Yaskawa INFORM job: pointsclTRJ2.JBI

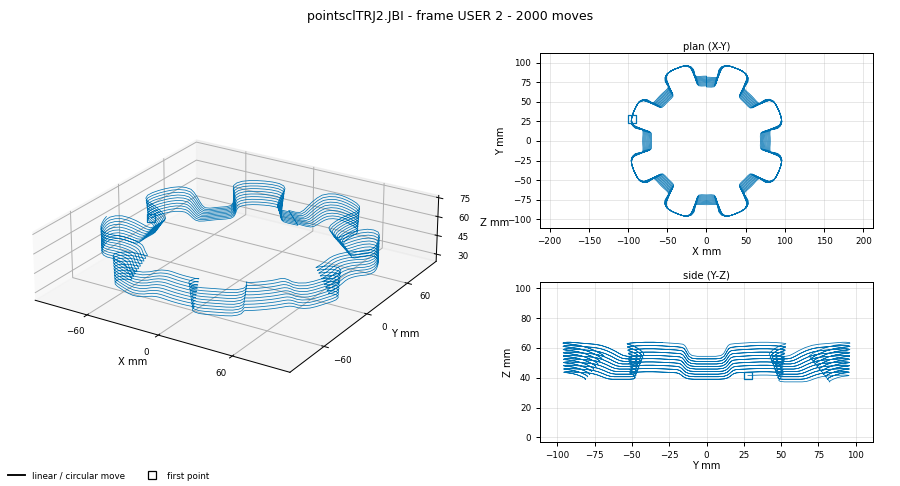
[picture p0: tool path of pointsclTRJ2.JBI in frame USER 2, 2000 of 2000 moves have a stored position in this frame; points joined in program order, loops and branches not executed]
/JOB
//NAME pointsclTRJ2
//POS
///NPOS 2000,0,0,0,0,0
///USER 2
///TOOL 1
///POSTYPE USER
///RECTAN
///RCONF 1,0,0,0,0,0,0,0,0,0,0,0,0,0,0,0,0,0,0,0,0,0,0,0
C00000=-95.500,27.752,41.515,166.5415,13.7835,0.0000
C00001=-94.679,31.992,41.678,168.5942,9.8161,0.0000
C00002=-93.214,36.189,41.785,170.1405,7.6437,0.0000
C00003=-91.502,40.323,41.785,-167.6355,-1.4870,0.0000
C00004=-89.570,44.326,41.678,-165.0261,-0.9876,0.0000
C00005=-87.153,47.905,41.515,-160.8334,0.4949,0.0000
C00006=-83.964,50.341,41.355,-155.1452,4.3197,0.0000
C00007=-80.606,51.270,41.159,-151.1279,10.7556,0.0000
C00008=-77.545,50.645,40.789,-149.8656,15.0064,0.0000
C00009=-74.511,49.565,40.048,-149.4700,17.9765,0.0000
C00010=-71.724,48.673,39.090,-149.4755,20.2620,0.0000
C00011=-69.261,48.447,38.165,-149.7708,22.3484,0.0000
C00012=-66.868,49.465,37.495,-150.5123,24.7951,0.0000
C00013=-64.059,52.288,37.229,-151.9366,27.5294,0.0000
C00014=-61.349,55.398,37.217,-151.9559,27.7386,0.0000
C00015=-58.451,58.451,37.225,-150.5381,26.1896,0.0000
C00016=-55.398,61.349,37.217,-149.2124,24.5903,0.0000
C00017=-52.288,64.059,37.229,-149.4318,24.6574,0.0000
C00018=-49.465,66.868,37.495,-152.0451,26.5426,0.0000
C00019=-48.447,69.261,38.165,-154.5539,27.7518,0.0000
C00020=-48.673,71.724,39.090,-156.8022,28.4553,0.0000
C00021=-49.565,74.511,40.048,-159.3588,28.8937,0.0000
C00022=-50.645,77.545,40.789,-162.7782,29.0063,0.0000
C00023=-51.270,80.606,41.159,-167.7607,28.3185,0.0000
C00024=-50.341,83.964,41.355,-175.2412,24.7794,0.0000
C00025=-47.905,87.153,41.515,-179.4760,19.1659,0.0000
C00026=-44.326,89.570,41.678,178.9776,14.9716,0.0000
C00027=-40.323,91.502,41.785,178.4777,12.3603,0.0000
C00028=-36.189,93.214,41.785,-172.2431,-9.7711,0.0000
C00029=-31.992,94.679,41.678,-169.9901,-11.2367,0.0000
C00030=-27.752,95.500,41.515,-165.8427,-13.0639,0.0000
C00031=-23.775,94.968,41.355,-158.8727,-14.0699,0.0000
C00032=-20.743,93.250,41.159,-151.4855,-11.7399,0.0000
C00033=-19.021,90.644,40.789,-147.8038,-9.1945,0.0000
C00034=-17.640,87.735,40.048,-145.6522,-7.0900,0.0000
C00035=-16.299,85.134,39.090,-144.2478,-5.2806,0.0000
C00036=-14.718,83.232,38.165,-143.1858,-3.4622,0.0000
C00037=-12.305,82.260,37.495,-142.2198,-1.1140,0.0000
C00038=-8.324,82.270,37.229,-141.5279,1.8234,0.0000
C00039=-4.208,82.553,37.217,-141.4104,1.9981,0.0000
C00040=0.000,82.662,37.225,-141.3795,0.0003,0.0000
C00041=0.000,81.307,38.958,-141.1409,0.0002,0.0000
C00042=4.084,81.202,38.949,-141.1716,-1.9954,0.0000
C00043=8.115,80.931,38.962,-141.2889,-1.7381,0.0000
C00044=12.050,80.963,39.253,-141.9942,1.3169,0.0000
C00045=14.402,82.041,39.987,-142.9610,3.6876,0.0000
C00046=15.932,84.113,41.004,-144.0223,5.5238,0.0000
C00047=17.234,86.943,42.060,-145.4570,7.3915,0.0000
C00048=18.580,90.119,42.880,-147.7223,9.6046,0.0000
C00049=20.259,92.987,43.289,-151.7341,12.2844,0.0000
C00050=23.317,94.913,43.506,-160.1091,14.4794,0.0000
C00051=27.389,95.566,43.684,-167.4562,12.7995,0.0000
C00052=31.762,94.755,43.864,-171.4202,10.6129,0.0000
C00053=36.110,93.244,43.984,-173.4230,9.0647,0.0000
C00054=40.400,91.468,43.984,178.1652,-11.0336,0.0000
C00055=44.543,89.461,43.864,178.4356,-13.5277,0.0000
C00056=48.209,86.942,43.684,179.5849,-17.8430,0.0000
C00057=50.626,83.601,43.506,-176.4717,-24.1883,0.0000
C00058=51.426,80.077,43.289,-168.3941,-28.5314,0.0000
C00059=50.586,76.861,42.880,-163.0330,-29.3601,0.0000
C00060=49.291,73.664,42.060,-159.4239,-29.2475,0.0000
C00061=48.211,70.742,41.004,-156.7894,-28.7861,0.0000
C00062=47.828,68.195,39.987,-154.5220,-28.0686,0.0000
C00063=48.729,65.770,39.253,-151.9898,-26.8420,0.0000
C00064=51.488,62.965,38.962,-149.2803,-24.8706,0.0000
C00065=54.531,60.307,38.949,-149.0055,-24.7373,0.0000
C00066=57.493,57.493,38.958,-150.3287,-26.3368,0.0000
C00067=60.306,54.531,38.949,-151.7425,-27.8849,0.0000
C00068=62.965,51.488,38.962,-151.6647,-27.6101,0.0000
C00069=65.770,48.729,39.253,-150.1785,-24.7729,0.0000
C00070=68.195,47.828,39.987,-149.4302,-22.3072,0.0000
C00071=70.742,48.211,41.004,-149.1281,-20.2070,0.0000
C00072=73.664,49.291,42.060,-149.1154,-17.8577,0.0000
C00073=76.861,50.586,42.880,-149.5380,-14.7348,0.0000
C00074=80.077,51.426,43.289,-150.9692,-10.1806,0.0000
C00075=83.601,50.626,43.506,-155.7711,-3.2182,0.0000
C00076=86.942,48.209,43.684,-162.1566,0.3951,0.0000
C00077=89.461,44.543,43.864,-166.4674,1.5210,0.0000
C00078=91.468,40.400,43.984,-168.9609,1.8009,0.0000
C00079=93.244,36.110,43.984,170.8762,-6.4945,0.0000
C00080=94.755,31.762,43.864,169.2698,-8.4320,0.0000
C00081=95.566,27.389,43.684,166.8982,-12.2272,0.0000
C00082=94.913,23.317,43.506,164.6442,-19.2338,0.0000
C00083=92.987,20.259,43.289,166.1133,-27.5629,0.0000
C00084=90.119,18.580,42.880,168.6818,-31.7718,0.0000
C00085=86.943,17.234,42.060,171.0499,-34.2159,0.0000
C00086=84.113,15.932,41.004,173.1852,-35.7848,0.0000
C00087=82.041,14.402,39.987,175.3839,-36.9495,0.0000
C00088=80.963,12.050,39.253,178.3288,-37.9940,0.0000
C00089=80.931,8.115,38.962,-177.7730,-38.6900,0.0000
C00090=81.202,4.084,38.949,-177.4393,-38.8004,0.0000
C00091=81.307,0.000,38.958,179.9997,-38.8591,0.0000
C00092=81.202,-4.084,38.949,177.4397,-38.8005,0.0000
C00093=80.931,-8.116,38.962,177.7742,-38.6899,0.0000
C00094=80.963,-12.050,39.253,-178.3283,-37.9939,0.0000
C00095=82.041,-14.402,39.987,-175.3840,-36.9495,0.0000
C00096=84.113,-15.932,41.004,-173.1855,-35.7848,0.0000
C00097=86.943,-17.234,42.060,-171.0504,-34.2160,0.0000
C00098=90.119,-18.580,42.880,-168.6823,-31.7720,0.0000
C00099=92.987,-20.259,43.289,-166.1135,-27.5630,0.0000
C00100=94.913,-23.317,43.506,-164.6442,-19.2338,0.0000
C00101=95.566,-27.389,43.684,-166.8982,-12.2272,0.0000
C00102=94.755,-31.762,43.864,-169.2698,-8.4320,0.0000
C00103=93.244,-36.110,43.984,-170.8762,-6.4945,0.0000
C00104=91.468,-40.400,43.984,168.9609,1.8009,0.0000
C00105=89.461,-44.543,43.864,166.4674,1.5210,0.0000
C00106=86.942,-48.209,43.684,162.1566,0.3951,0.0000
C00107=83.601,-50.626,43.506,155.7711,-3.2182,0.0000
C00108=80.077,-51.426,43.289,150.9692,-10.1803,0.0000
C00109=76.861,-50.586,42.880,149.5378,-14.7344,0.0000
C00110=73.664,-49.291,42.060,149.1152,-17.8573,0.0000
C00111=70.742,-48.211,41.004,149.1280,-20.2068,0.0000
C00112=68.195,-47.828,39.987,149.4301,-22.3071,0.0000
C00113=65.770,-48.729,39.253,150.1787,-24.7733,0.0000
C00114=62.965,-51.488,38.962,151.6652,-27.6109,0.0000
C00115=60.307,-54.531,38.949,151.7428,-27.8851,0.0000
C00116=57.493,-57.493,38.958,150.3283,-26.3364,0.0000
C00117=54.531,-60.306,38.949,149.0057,-24.7376,0.0000
C00118=51.488,-62.965,38.962,149.2810,-24.8713,0.0000
C00119=48.729,-65.770,39.253,151.9902,-26.8422,0.0000
C00120=47.828,-68.195,39.987,154.5219,-28.0685,0.0000
C00121=48.211,-70.742,41.004,156.7892,-28.7859,0.0000
C00122=49.291,-73.664,42.060,159.4235,-29.2473,0.0000
C00123=50.586,-76.861,42.880,163.0325,-29.3600,0.0000
C00124=51.426,-80.077,43.289,168.3938,-28.5314,0.0000
C00125=50.626,-83.601,43.506,176.4717,-24.1883,0.0000
C00126=48.209,-86.942,43.684,-179.5849,-17.8430,0.0000
C00127=44.543,-89.461,43.864,-178.4356,-13.5277,0.0000
C00128=40.400,-91.468,43.984,-178.1652,-11.0336,0.0000
C00129=36.110,-93.244,43.984,173.4230,9.0647,0.0000
C00130=31.762,-94.755,43.864,171.4202,10.6129,0.0000
C00131=27.389,-95.566,43.684,167.4562,12.7995,0.0000
C00132=23.317,-94.913,43.506,160.1091,14.4794,0.0000
C00133=20.259,-92.987,43.289,151.7341,12.2844,0.0000
C00134=18.580,-90.119,42.880,147.7223,9.6046,0.0000
C00135=17.234,-86.943,42.060,145.4570,7.3915,0.0000
C00136=15.932,-84.113,41.004,144.0223,5.5238,0.0000
C00137=14.402,-82.041,39.987,142.9610,3.6876,0.0000
C00138=12.050,-80.963,39.253,141.9942,1.3169,0.0000
C00139=8.115,-80.931,38.962,141.2889,-1.7381,0.0000
C00140=4.084,-81.202,38.949,141.1716,-1.9954,0.0000
C00141=0.000,-81.307,38.958,141.1409,0.0002,0.0000
C00142=0.000,-81.307,38.958,141.1409,0.0002,0.0000
C00143=-4.084,-81.202,38.949,141.1716,1.9951,0.0000
C00144=-8.116,-80.931,38.962,141.2890,1.7371,0.0000
C00145=-12.050,-80.963,39.253,141.9943,-1.3173,0.0000
C00146=-14.402,-82.041,39.987,142.9611,-3.6875,0.0000
C00147=-15.932,-84.113,41.004,144.0223,-5.5235,0.0000
C00148=-17.234,-86.943,42.060,145.4569,-7.3911,0.0000
C00149=-18.580,-90.119,42.880,147.7222,-9.6042,0.0000
C00150=-20.259,-92.987,43.289,151.7339,-12.2842,0.0000
C00151=-23.317,-94.913,43.506,160.1091,-14.4794,0.0000
C00152=-27.389,-95.566,43.684,167.4562,-12.7995,0.0000
C00153=-31.762,-94.755,43.864,171.4202,-10.6129,0.0000
C00154=-36.110,-93.244,43.984,173.4230,-9.0647,0.0000
C00155=-40.400,-91.468,43.984,-178.1652,11.0336,0.0000
C00156=-44.543,-89.461,43.864,-178.4356,13.5277,0.0000
C00157=-48.209,-86.942,43.684,-179.5849,17.8430,0.0000
C00158=-50.626,-83.601,43.506,176.4717,24.1883,0.0000
C00159=-51.426,-80.077,43.289,168.3941,28.5314,0.0000
C00160=-50.586,-76.861,42.880,163.0330,29.3601,0.0000
C00161=-49.291,-73.664,42.060,159.4239,29.2475,0.0000
C00162=-48.211,-70.742,41.004,156.7894,28.7861,0.0000
C00163=-47.828,-68.195,39.987,154.5220,28.0686,0.0000
C00164=-48.729,-65.770,39.253,151.9898,26.8420,0.0000
C00165=-51.488,-62.965,38.962,149.2803,24.8706,0.0000
C00166=-54.531,-60.307,38.949,149.0055,24.7373,0.0000
C00167=-57.493,-57.493,38.958,150.3287,26.3368,0.0000
C00168=-60.306,-54.531,38.949,151.7425,27.8849,0.0000
C00169=-62.965,-51.488,38.962,151.6647,27.6101,0.0000
C00170=-65.770,-48.729,39.253,150.1785,24.7729,0.0000
C00171=-68.195,-47.828,39.987,149.4302,22.3072,0.0000
C00172=-70.742,-48.211,41.004,149.1281,20.2070,0.0000
C00173=-73.664,-49.291,42.060,149.1154,17.8577,0.0000
C00174=-76.861,-50.586,42.880,149.5380,14.7348,0.0000
C00175=-80.077,-51.426,43.289,150.9692,10.1806,0.0000
C00176=-83.601,-50.626,43.506,155.7711,3.2182,0.0000
C00177=-86.942,-48.209,43.684,162.1566,-0.3951,0.0000
C00178=-89.461,-44.543,43.864,166.4674,-1.5210,0.0000
C00179=-91.468,-40.400,43.984,168.9609,-1.8009,0.0000
C00180=-93.244,-36.110,43.984,-170.8762,6.4945,0.0000
C00181=-94.755,-31.762,43.864,-169.2698,8.4320,0.0000
C00182=-95.566,-27.389,43.684,-166.8982,12.2272,0.0000
C00183=-94.913,-23.317,43.506,-164.6442,19.2338,0.0000
C00184=-92.987,-20.259,43.289,-166.1133,27.5629,0.0000
C00185=-90.119,-18.580,42.880,-168.6818,31.7718,0.0000
C00186=-86.943,-17.234,42.060,-171.0499,34.2159,0.0000
C00187=-84.113,-15.932,41.004,-173.1852,35.7848,0.0000
C00188=-82.041,-14.402,39.987,-175.3839,36.9495,0.0000
C00189=-80.963,-12.050,39.253,-178.3288,37.9940,0.0000
C00190=-80.931,-8.115,38.962,177.7730,38.6900,0.0000
C00191=-81.202,-4.084,38.949,177.4393,38.8004,0.0000
C00192=-81.307,0.000,38.958,-179.9997,38.8591,0.0000
C00193=-81.202,4.084,38.949,-177.4397,38.8005,0.0000
C00194=-80.931,8.116,38.962,-177.7742,38.6899,0.0000
C00195=-80.963,12.050,39.253,178.3283,37.9939,0.0000
C00196=-82.041,14.402,39.987,175.3840,36.9495,0.0000
C00197=-84.113,15.932,41.004,173.1855,35.7848,0.0000
C00198=-86.943,17.234,42.060,171.0504,34.2160,0.0000
C00199=-90.119,18.580,42.880,168.6823,31.7720,0.0000
C00200=-92.987,20.259,43.289,166.1135,27.5630,0.0000
C00201=-94.913,23.317,43.506,164.6442,19.2338,0.0000
C00202=-95.566,27.389,43.684,166.8982,12.2272,0.0000
C00203=-94.755,31.762,43.864,169.2698,8.4320,0.0000
C00204=-93.244,36.110,43.984,170.8762,6.4945,0.0000
C00205=-91.468,40.400,43.984,-168.9609,-1.8009,0.0000
C00206=-89.461,44.543,43.864,-166.4674,-1.5210,0.0000
C00207=-86.942,48.209,43.684,-162.1566,-0.3951,0.0000
C00208=-83.601,50.626,43.506,-155.7711,3.2182,0.0000
C00209=-80.077,51.426,43.289,-150.9692,10.1803,0.0000
C00210=-76.861,50.586,42.880,-149.5378,14.7344,0.0000
C00211=-73.664,49.291,42.060,-149.1152,17.8573,0.0000
C00212=-70.742,48.211,41.004,-149.1280,20.2068,0.0000
C00213=-68.195,47.828,39.987,-149.4301,22.3071,0.0000
C00214=-65.770,48.729,39.253,-150.1787,24.7733,0.0000
C00215=-62.965,51.488,38.962,-151.6652,27.6109,0.0000
C00216=-60.307,54.531,38.949,-151.7428,27.8851,0.0000
C00217=-57.493,57.493,38.958,-150.3283,26.3364,0.0000
C00218=-54.531,60.306,38.949,-149.0057,24.7376,0.0000
C00219=-51.488,62.965,38.962,-149.2810,24.8713,0.0000
C00220=-48.729,65.770,39.253,-151.9902,26.8422,0.0000
C00221=-47.828,68.195,39.987,-154.5219,28.0685,0.0000
C00222=-48.211,70.742,41.004,-156.7892,28.7859,0.0000
C00223=-49.291,73.664,42.060,-159.4235,29.2473,0.0000
C00224=-50.586,76.861,42.880,-163.0325,29.3600,0.0000
C00225=-51.426,80.077,43.289,-168.3938,28.5314,0.0000
C00226=-50.626,83.601,43.506,-176.4717,24.1883,0.0000
C00227=-48.209,86.942,43.684,179.5849,17.8430,0.0000
C00228=-44.543,89.461,43.864,178.4356,13.5277,0.0000
C00229=-40.400,91.468,43.984,178.1652,11.0336,0.0000
C00230=-36.110,93.244,43.984,-173.4230,-9.0647,0.0000
C00231=-31.762,94.755,43.864,-171.4202,-10.6129,0.0000
C00232=-27.389,95.566,43.684,-167.4562,-12.7995,0.0000
C00233=-23.317,94.913,43.506,-160.1091,-14.4794,0.0000
C00234=-20.259,92.987,43.289,-151.7339,-12.2842,0.0000
C00235=-18.580,90.119,42.880,-147.7222,-9.6042,0.0000
C00236=-17.234,86.943,42.060,-145.4569,-7.3911,0.0000
C00237=-15.932,84.113,41.004,-144.0223,-5.5235,0.0000
C00238=-14.402,82.041,39.987,-142.9611,-3.6875,0.0000
C00239=-12.050,80.963,39.253,-141.9943,-1.3173,0.0000
C00240=-8.116,80.931,38.962,-141.2890,1.7371,0.0000
C00241=-4.084,81.202,38.949,-141.1716,1.9951,0.0000
C00242=0.000,81.307,38.958,-141.1409,0.0002,0.0000
C00243=0.000,79.940,40.681,-140.9575,0.0002,0.0000
C00244=3.959,79.840,40.672,-140.9880,-1.9887,0.0000
C00245=7.905,79.580,40.686,-141.1052,-1.6534,0.0000
C00246=11.791,79.654,41.003,-141.8234,1.5070,0.0000
C00247=14.083,80.839,41.802,-142.7891,3.8920,0.0000
C00248=15.561,83.082,42.912,-143.8479,5.7437,0.0000
C00249=16.825,86.143,44.068,-145.3137,7.6721,0.0000
C00250=18.134,89.588,44.968,-147.7068,10.0045,0.0000
C00251=19.771,92.721,45.418,-152.1169,12.8313,0.0000
C00252=22.856,94.857,45.657,-161.6285,14.7239,0.0000
C00253=27.022,95.633,45.852,-169.2186,12.2388,0.0000
C00254=31.529,94.831,46.051,-172.8727,9.7455,0.0000
C00255=36.031,93.275,46.182,-174.5815,8.1817,0.0000
C00256=40.478,91.433,46.182,177.9926,-9.5974,0.0000
C00257=44.762,89.350,46.051,178.0542,-11.8975,0.0000
C00258=48.515,86.730,45.852,178.7689,-16.2103,0.0000
C00259=50.913,83.236,45.657,-177.7648,-23.2825,0.0000
C00260=51.583,79.544,45.418,-169.1361,-28.6508,0.0000
C00261=50.526,76.172,44.968,-163.3358,-29.6613,0.0000
C00262=49.015,72.810,44.068,-159.5177,-29.5512,0.0000
C00263=47.744,69.752,42.912,-156.8033,-29.0660,0.0000
C00264=47.203,67.120,41.802,-154.5207,-28.3354,0.0000
C00265=47.986,64.662,41.003,-151.9734,-27.0971,0.0000
C00266=50.682,61.862,40.686,-149.1762,-25.0495,0.0000
C00267=53.655,59.255,40.672,-148.8492,-24.8539,0.0000
C00268=56.526,56.526,40.681,-150.1670,-26.4494,0.0000
C00269=59.255,53.656,40.672,-151.5753,-27.9941,0.0000
C00270=61.862,50.682,40.686,-151.4429,-27.6579,0.0000
C00271=64.662,47.986,41.003,-149.9017,-24.7273,0.0000
C00272=67.120,47.203,41.802,-149.1486,-22.2497,0.0000
C00273=69.752,47.744,42.912,-148.8387,-20.1383,0.0000
C00274=72.810,49.015,44.068,-148.8172,-17.7224,0.0000
C00275=76.172,50.526,44.968,-149.2703,-14.4298,0.0000
C00276=79.544,51.583,45.418,-150.9111,-9.5207,0.0000
C00277=83.236,50.913,45.657,-156.7016,-2.0531,0.0000
C00278=86.730,48.515,45.852,-163.7862,1.1821,0.0000
C00279=89.350,44.762,46.051,-168.0959,1.9040,0.0000
C00280=91.433,40.478,46.182,-170.3968,1.9793,0.0000
C00281=93.275,36.031,46.182,171.7820,-5.3632,0.0000
C00282=94.831,31.529,46.051,170.1801,-7.0240,0.0000
C00283=95.633,27.022,45.852,167.5481,-10.5335,0.0000
C00284=94.857,22.856,45.657,164.5223,-17.7478,0.0000
C00285=92.721,19.771,45.418,165.5501,-27.1287,0.0000
C00286=89.588,18.134,44.968,168.2123,-31.7442,0.0000
C00287=86.143,16.825,44.068,170.6962,-34.3321,0.0000
C00288=83.082,15.561,42.912,172.8993,-35.9422,0.0000
C00289=80.839,14.083,41.802,175.1175,-37.1107,0.0000
C00290=79.654,11.791,41.003,178.0832,-38.1610,0.0000
C00291=79.580,7.905,40.686,-177.8761,-38.8756,0.0000
C00292=79.840,3.959,40.672,-177.4412,-38.9841,0.0000
C00293=79.940,0.000,40.681,179.9998,-39.0425,0.0000
C00294=79.840,-3.959,40.672,177.4416,-38.9841,0.0000
C00295=79.580,-7.905,40.686,177.8773,-38.8755,0.0000
C00296=79.654,-11.792,41.003,-178.0827,-38.1609,0.0000
C00297=80.839,-14.083,41.802,-175.1176,-37.1106,0.0000
C00298=83.082,-15.561,42.912,-172.8996,-35.9423,0.0000
C00299=86.143,-16.825,44.068,-170.6967,-34.3323,0.0000
C00300=89.588,-18.134,44.968,-168.2127,-31.7445,0.0000
C00301=92.721,-19.771,45.418,-165.5503,-27.1290,0.0000
C00302=94.857,-22.856,45.657,-164.5223,-17.7478,0.0000
C00303=95.633,-27.022,45.852,-167.5481,-10.5335,0.0000
C00304=94.831,-31.529,46.051,-170.1801,-7.0240,0.0000
C00305=93.275,-36.031,46.182,-171.7820,-5.3632,0.0000
C00306=91.433,-40.478,46.182,170.3968,1.9793,0.0000
C00307=89.350,-44.762,46.051,168.0959,1.9040,0.0000
C00308=86.730,-48.515,45.852,163.7862,1.1821,0.0000
C00309=83.236,-50.913,45.657,156.7016,-2.0531,0.0000
C00310=79.544,-51.583,45.418,150.9111,-9.5204,0.0000
C00311=76.172,-50.526,44.968,149.2702,-14.4293,0.0000
C00312=72.810,-49.015,44.068,148.8170,-17.7220,0.0000
C00313=69.752,-47.744,42.912,148.8386,-20.1381,0.0000
C00314=67.120,-47.203,41.802,149.1485,-22.2496,0.0000
C00315=64.662,-47.986,41.003,149.9019,-24.7276,0.0000
C00316=61.862,-50.682,40.686,151.4435,-27.6587,0.0000
C00317=59.255,-53.655,40.672,151.5755,-27.9942,0.0000
C00318=56.526,-56.526,40.681,150.1668,-26.4491,0.0000
C00319=53.656,-59.255,40.672,148.8493,-24.8541,0.0000
C00320=50.682,-61.862,40.686,149.1770,-25.0502,0.0000
C00321=47.986,-64.662,41.003,151.9738,-27.0973,0.0000
C00322=47.203,-67.120,41.802,154.5206,-28.3353,0.0000
C00323=47.744,-69.752,42.912,156.8030,-29.0658,0.0000
C00324=49.015,-72.810,44.068,159.5173,-29.5510,0.0000
C00325=50.526,-76.172,44.968,163.3354,-29.6611,0.0000
C00326=51.583,-79.544,45.418,169.1358,-28.6508,0.0000
C00327=50.913,-83.236,45.657,177.7648,-23.2825,0.0000
C00328=48.515,-86.730,45.852,-178.7689,-16.2103,0.0000
C00329=44.762,-89.350,46.051,-178.0542,-11.8975,0.0000
C00330=40.478,-91.433,46.182,-177.9926,-9.5974,0.0000
C00331=36.031,-93.275,46.182,174.5815,8.1817,0.0000
C00332=31.529,-94.831,46.051,172.8727,9.7455,0.0000
C00333=27.022,-95.633,45.852,169.2186,12.2388,0.0000
C00334=22.856,-94.857,45.657,161.6285,14.7239,0.0000
C00335=19.771,-92.721,45.418,152.1169,12.8313,0.0000
C00336=18.134,-89.588,44.968,147.7068,10.0045,0.0000
C00337=16.825,-86.143,44.068,145.3137,7.6721,0.0000
C00338=15.561,-83.082,42.912,143.8479,5.7437,0.0000
C00339=14.083,-80.839,41.802,142.7891,3.8920,0.0000
C00340=11.791,-79.654,41.003,141.8234,1.5070,0.0000
C00341=7.905,-79.580,40.686,141.1052,-1.6534,0.0000
C00342=3.959,-79.840,40.672,140.9880,-1.9887,0.0000
C00343=0.000,-79.940,40.681,140.9575,0.0002,0.0000
C00344=0.000,-79.940,40.681,140.9575,0.0002,0.0000
C00345=-3.959,-79.840,40.672,140.9879,1.9885,0.0000
C00346=-7.905,-79.580,40.686,141.1053,1.6524,0.0000
C00347=-11.792,-79.654,41.003,141.8235,-1.5075,0.0000
C00348=-14.083,-80.839,41.802,142.7891,-3.8919,0.0000
C00349=-15.561,-83.082,42.912,143.8478,-5.7435,0.0000
C00350=-16.825,-86.143,44.068,145.3136,-7.6717,0.0000
C00351=-18.134,-89.588,44.968,147.7066,-10.0041,0.0000
C00352=-19.771,-92.721,45.418,152.1166,-12.8311,0.0000
C00353=-22.856,-94.857,45.657,161.6285,-14.7239,0.0000
C00354=-27.022,-95.633,45.852,169.2186,-12.2388,0.0000
C00355=-31.529,-94.831,46.051,172.8727,-9.7455,0.0000
C00356=-36.031,-93.275,46.182,174.5815,-8.1817,0.0000
C00357=-40.478,-91.433,46.182,-177.9926,9.5974,0.0000
C00358=-44.762,-89.350,46.051,-178.0542,11.8975,0.0000
C00359=-48.515,-86.730,45.852,-178.7689,16.2103,0.0000
C00360=-50.913,-83.236,45.657,177.7648,23.2825,0.0000
C00361=-51.583,-79.544,45.418,169.1361,28.6508,0.0000
C00362=-50.526,-76.172,44.968,163.3358,29.6613,0.0000
C00363=-49.015,-72.810,44.068,159.5177,29.5512,0.0000
C00364=-47.744,-69.752,42.912,156.8033,29.0660,0.0000
C00365=-47.203,-67.120,41.802,154.5207,28.3354,0.0000
C00366=-47.986,-64.662,41.003,151.9734,27.0971,0.0000
C00367=-50.682,-61.862,40.686,149.1762,25.0495,0.0000
C00368=-53.655,-59.255,40.672,148.8492,24.8539,0.0000
C00369=-56.526,-56.526,40.681,150.1670,26.4494,0.0000
C00370=-59.255,-53.656,40.672,151.5753,27.9941,0.0000
C00371=-61.862,-50.682,40.686,151.4429,27.6579,0.0000
C00372=-64.662,-47.986,41.003,149.9017,24.7273,0.0000
C00373=-67.120,-47.203,41.802,149.1486,22.2497,0.0000
C00374=-69.752,-47.744,42.912,148.8387,20.1383,0.0000
C00375=-72.810,-49.015,44.068,148.8172,17.7224,0.0000
C00376=-76.172,-50.526,44.968,149.2703,14.4298,0.0000
C00377=-79.544,-51.583,45.418,150.9111,9.5207,0.0000
C00378=-83.236,-50.913,45.657,156.7016,2.0531,0.0000
C00379=-86.730,-48.515,45.852,163.7862,-1.1821,0.0000
C00380=-89.350,-44.762,46.051,168.0959,-1.9040,0.0000
C00381=-91.433,-40.478,46.182,170.3968,-1.9793,0.0000
C00382=-93.275,-36.031,46.182,-171.7820,5.3632,0.0000
C00383=-94.831,-31.529,46.051,-170.1801,7.0240,0.0000
C00384=-95.633,-27.022,45.852,-167.5481,10.5335,0.0000
C00385=-94.857,-22.856,45.657,-164.5223,17.7478,0.0000
C00386=-92.721,-19.771,45.418,-165.5501,27.1287,0.0000
C00387=-89.588,-18.134,44.968,-168.2123,31.7442,0.0000
C00388=-86.143,-16.825,44.068,-170.6962,34.3321,0.0000
C00389=-83.082,-15.561,42.912,-172.8993,35.9422,0.0000
C00390=-80.839,-14.083,41.802,-175.1175,37.1107,0.0000
C00391=-79.654,-11.791,41.003,-178.0832,38.1610,0.0000
C00392=-79.580,-7.905,40.686,177.8761,38.8756,0.0000
C00393=-79.840,-3.959,40.672,177.4412,38.9841,0.0000
C00394=-79.940,0.000,40.681,-179.9998,39.0425,0.0000
C00395=-79.840,3.959,40.672,-177.4416,38.9841,0.0000
C00396=-79.580,7.905,40.686,-177.8773,38.8755,0.0000
C00397=-79.654,11.792,41.003,178.0827,38.1609,0.0000
C00398=-80.839,14.083,41.802,175.1176,37.1106,0.0000
C00399=-83.082,15.561,42.912,172.8996,35.9423,0.0000
C00400=-86.143,16.825,44.068,170.6967,34.3323,0.0000
C00401=-89.588,18.134,44.968,168.2127,31.7445,0.0000
C00402=-92.721,19.771,45.418,165.5503,27.1290,0.0000
C00403=-94.857,22.856,45.657,164.5223,17.7478,0.0000
C00404=-95.633,27.022,45.852,167.5481,10.5335,0.0000
C00405=-94.831,31.529,46.051,170.1801,7.0240,0.0000
C00406=-93.275,36.031,46.182,171.7820,5.3632,0.0000
C00407=-91.433,40.478,46.182,-170.3968,-1.9793,0.0000
C00408=-89.350,44.762,46.051,-168.0959,-1.9040,0.0000
C00409=-86.730,48.515,45.852,-163.7862,-1.1821,0.0000
C00410=-83.236,50.913,45.657,-156.7016,2.0531,0.0000
C00411=-79.544,51.583,45.418,-150.9111,9.5204,0.0000
C00412=-76.172,50.526,44.968,-149.2702,14.4293,0.0000
C00413=-72.810,49.015,44.068,-148.8170,17.7220,0.0000
C00414=-69.752,47.744,42.912,-148.8386,20.1381,0.0000
C00415=-67.120,47.203,41.802,-149.1485,22.2496,0.0000
C00416=-64.662,47.986,41.003,-149.9019,24.7276,0.0000
C00417=-61.862,50.682,40.686,-151.4435,27.6587,0.0000
C00418=-59.255,53.655,40.672,-151.5755,27.9942,0.0000
C00419=-56.526,56.526,40.681,-150.1668,26.4491,0.0000
C00420=-53.656,59.255,40.672,-148.8493,24.8541,0.0000
C00421=-50.682,61.862,40.686,-149.1770,25.0502,0.0000
C00422=-47.986,64.662,41.003,-151.9738,27.0973,0.0000
C00423=-47.203,67.120,41.802,-154.5206,28.3353,0.0000
C00424=-47.744,69.752,42.912,-156.8030,29.0658,0.0000
C00425=-49.015,72.810,44.068,-159.5173,29.5510,0.0000
C00426=-50.526,76.172,44.968,-163.3354,29.6611,0.0000
C00427=-51.583,79.544,45.418,-169.1358,28.6508,0.0000
C00428=-50.913,83.236,45.657,-177.7648,23.2825,0.0000
C00429=-48.515,86.730,45.852,178.7689,16.2103,0.0000
C00430=-44.762,89.350,46.051,178.0542,11.8975,0.0000
C00431=-40.478,91.433,46.182,177.9926,9.5974,0.0000
C00432=-36.031,93.275,46.182,-174.5815,-8.1817,0.0000
C00433=-31.529,94.831,46.051,-172.8727,-9.7455,0.0000
C00434=-27.022,95.633,45.852,-169.2186,-12.2388,0.0000
C00435=-22.856,94.857,45.657,-161.6285,-14.7239,0.0000
C00436=-19.771,92.721,45.418,-152.1166,-12.8311,0.0000
C00437=-18.134,89.588,44.968,-147.7066,-10.0041,0.0000
C00438=-16.825,86.143,44.068,-145.3136,-7.6717,0.0000
C00439=-15.561,83.082,42.912,-143.8478,-5.7435,0.0000
C00440=-14.083,80.839,41.802,-142.7891,-3.8919,0.0000
C00441=-11.792,79.654,41.003,-141.8235,-1.5075,0.0000
C00442=-7.905,79.580,40.686,-141.1053,1.6524,0.0000
C00443=-3.959,79.840,40.672,-140.9879,1.9885,0.0000
C00444=0.000,79.940,40.681,-140.9575,0.0002,0.0000
C00445=0.000,78.562,42.397,-140.8266,0.0001,0.0000
C00446=3.833,78.467,42.387,-140.8567,-1.9786,0.0000
C00447=7.694,78.220,42.402,-140.9739,-1.5709,0.0000
C00448=11.532,78.336,42.745,-141.7044,1.6835,0.0000
C00449=13.762,79.628,43.611,-142.6667,4.0757,0.0000
C00450=15.189,82.045,44.816,-143.7214,5.9414,0.0000
C00451=16.414,85.339,46.074,-145.2199,7.9339,0.0000
C00452=17.687,89.056,47.055,-147.7591,10.3985,0.0000
C00453=19.281,92.454,47.546,-152.6596,13.3840,0.0000
C00454=22.392,94.802,47.807,-163.4548,14.7350,0.0000
C00455=26.654,95.700,48.020,-171.0751,11.3454,0.0000
C00456=31.296,94.909,48.237,-174.2977,8.6450,0.0000
C00457=35.952,93.306,48.381,-175.6864,7.1438,0.0000
C00458=40.555,91.399,48.381,177.9646,-8.0888,0.0000
C00459=44.981,89.240,48.237,177.8561,-10.1221,0.0000
C00460=48.823,86.517,48.020,178.1345,-14.2800,0.0000
C00461=51.201,82.869,47.807,-179.0798,-21.9992,0.0000
C00462=51.741,79.009,47.546,-170.0075,-28.6603,0.0000
C00463=50.465,75.478,47.055,-163.6915,-29.9114,0.0000
C00464=48.737,71.950,46.074,-159.6398,-29.8080,0.0000
C00465=47.275,68.755,44.816,-156.8422,-29.2978,0.0000
C00466=46.575,66.037,43.611,-154.5478,-28.5548,0.0000
C00467=47.238,63.546,42.745,-151.9928,-27.3092,0.0000
C00468=49.870,60.750,42.402,-149.1164,-25.1946,0.0000
C00469=52.774,58.195,42.387,-148.7408,-24.9413,0.0000
C00470=55.552,55.552,42.397,-150.0514,-26.5296,0.0000
C00471=58.195,52.774,42.387,-151.4518,-28.0677,0.0000
C00472=60.750,49.870,42.402,-151.2690,-27.6747,0.0000
C00473=63.546,47.238,42.745,-149.6793,-24.6603,0.0000
C00474=66.037,46.575,43.611,-148.9232,-22.1779,0.0000
C00475=68.755,47.275,44.816,-148.6044,-20.0576,0.0000
C00476=71.950,48.737,46.074,-148.5724,-17.5715,0.0000
C00477=75.478,50.465,47.055,-149.0612,-14.0880,0.0000
C00478=79.009,51.741,47.546,-150.9695,-8.7582,0.0000
C00479=82.869,51.201,47.807,-157.9982,-0.8532,0.0000
C00480=86.517,48.823,48.020,-165.7127,1.8078,0.0000
C00481=89.240,44.981,48.237,-169.8709,2.1105,0.0000
C00482=91.399,40.555,48.381,-171.9062,2.0151,0.0000
C00483=93.306,35.952,48.381,172.8361,-4.2800,0.0000
C00484=94.909,31.296,48.237,171.3126,-5.6373,0.0000
C00485=95.700,26.654,48.020,168.5192,-8.7492,0.0000
C00486=94.802,22.392,47.807,164.6580,-15.9863,0.0000
C00487=92.454,19.281,47.546,165.0047,-26.5387,0.0000
C00488=89.056,17.687,47.055,167.7588,-31.6493,0.0000
C00489=85.339,16.414,46.074,170.3698,-34.4000,0.0000
C00490=82.045,15.189,44.816,172.6440,-36.0530,0.0000
C00491=79.628,13.762,43.611,174.8791,-37.2229,0.0000
C00492=78.336,11.532,42.745,177.8553,-38.2761,0.0000
C00493=78.220,7.694,42.402,-177.9782,-39.0086,0.0000
C00494=78.467,3.833,42.387,-177.4495,-39.1155,0.0000
C00495=78.562,0.000,42.397,179.9998,-39.1734,0.0000
C00496=78.467,-3.833,42.387,177.4498,-39.1155,0.0000
C00497=78.220,-7.694,42.402,177.9795,-39.0085,0.0000
C00498=78.336,-11.532,42.745,-177.8547,-38.2760,0.0000
C00499=79.628,-13.762,43.611,-174.8791,-37.2228,0.0000
C00500=82.045,-15.189,44.816,-172.6443,-36.0530,0.0000
C00501=85.339,-16.414,46.074,-170.3703,-34.4002,0.0000
C00502=89.056,-17.687,47.055,-167.7593,-31.6496,0.0000
C00503=92.454,-19.281,47.546,-165.0050,-26.5390,0.0000
C00504=94.802,-22.392,47.807,-164.6580,-15.9863,0.0000
C00505=95.700,-26.654,48.020,-168.5192,-8.7492,0.0000
C00506=94.909,-31.296,48.237,-171.3126,-5.6373,0.0000
C00507=93.306,-35.952,48.381,-172.8361,-4.2800,0.0000
C00508=91.399,-40.555,48.381,171.9062,2.0151,0.0000
C00509=89.240,-44.981,48.237,169.8709,2.1105,0.0000
C00510=86.517,-48.823,48.020,165.7127,1.8078,0.0000
C00511=82.869,-51.201,47.807,157.9982,-0.8532,0.0000
C00512=79.009,-51.741,47.546,150.9696,-8.7579,0.0000
C00513=75.478,-50.465,47.055,149.0612,-14.0876,0.0000
C00514=71.950,-48.737,46.074,148.5722,-17.5711,0.0000
C00515=68.755,-47.275,44.816,148.6043,-20.0574,0.0000
C00516=66.037,-46.575,43.611,148.9231,-22.1779,0.0000
C00517=63.546,-47.238,42.745,149.6795,-24.6607,0.0000
C00518=60.750,-49.870,42.402,151.2696,-27.6755,0.0000
C00519=58.195,-52.774,42.387,151.4520,-28.0679,0.0000
C00520=55.552,-55.552,42.397,150.0512,-26.5294,0.0000
C00521=52.774,-58.195,42.387,148.7409,-24.9415,0.0000
C00522=49.870,-60.750,42.402,149.1172,-25.1953,0.0000
C00523=47.238,-63.546,42.745,151.9932,-27.3095,0.0000
C00524=46.575,-66.037,43.611,154.5477,-28.5547,0.0000
C00525=47.275,-68.755,44.816,156.8420,-29.2977,0.0000
C00526=48.737,-71.950,46.074,159.6394,-29.8078,0.0000
C00527=50.465,-75.478,47.055,163.6910,-29.9113,0.0000
C00528=51.741,-79.009,47.546,170.0072,-28.6603,0.0000
C00529=51.201,-82.869,47.807,179.0798,-21.9992,0.0000
C00530=48.823,-86.517,48.020,-178.1345,-14.2800,0.0000
C00531=44.981,-89.240,48.237,-177.8561,-10.1221,0.0000
C00532=40.555,-91.399,48.381,-177.9646,-8.0888,0.0000
C00533=35.952,-93.306,48.381,175.6864,7.1438,0.0000
C00534=31.296,-94.909,48.237,174.2977,8.6450,0.0000
C00535=26.654,-95.700,48.020,171.0751,11.3454,0.0000
C00536=22.392,-94.802,47.807,163.4548,14.7350,0.0000
C00537=19.281,-92.454,47.546,152.6596,13.3840,0.0000
C00538=17.687,-89.056,47.055,147.7591,10.3985,0.0000
C00539=16.414,-85.339,46.074,145.2199,7.9339,0.0000
C00540=15.189,-82.045,44.816,143.7214,5.9414,0.0000
C00541=13.762,-79.628,43.611,142.6667,4.0757,0.0000
C00542=11.532,-78.336,42.745,141.7044,1.6835,0.0000
C00543=7.694,-78.220,42.402,140.9739,-1.5709,0.0000
C00544=3.833,-78.467,42.387,140.8567,-1.9786,0.0000
C00545=0.000,-78.562,42.397,140.8266,0.0001,0.0000
C00546=0.000,-78.562,42.397,140.8266,0.0001,0.0000
C00547=-3.833,-78.467,42.387,140.8567,1.9784,0.0000
C00548=-7.694,-78.220,42.402,140.9740,1.5699,0.0000
C00549=-11.532,-78.336,42.745,141.7045,-1.6840,0.0000
C00550=-13.762,-79.628,43.611,142.6667,-4.0757,0.0000
C00551=-15.189,-82.045,44.816,143.7214,-5.9412,0.0000
C00552=-16.414,-85.339,46.074,145.2198,-7.9336,0.0000
C00553=-17.687,-89.056,47.055,147.7588,-10.3981,0.0000
C00554=-19.281,-92.454,47.546,152.6593,-13.3838,0.0000
C00555=-22.392,-94.802,47.807,163.4548,-14.7350,0.0000
C00556=-26.654,-95.700,48.020,171.0751,-11.3454,0.0000
C00557=-31.296,-94.909,48.237,174.2977,-8.6450,0.0000
C00558=-35.952,-93.306,48.381,175.6864,-7.1438,0.0000
C00559=-40.555,-91.399,48.381,-177.9646,8.0888,0.0000
C00560=-44.981,-89.240,48.237,-177.8561,10.1221,0.0000
C00561=-48.823,-86.517,48.020,-178.1345,14.2800,0.0000
C00562=-51.201,-82.869,47.807,179.0798,21.9992,0.0000
C00563=-51.741,-79.009,47.546,170.0075,28.6603,0.0000
C00564=-50.465,-75.478,47.055,163.6915,29.9114,0.0000
C00565=-48.737,-71.950,46.074,159.6398,29.8080,0.0000
C00566=-47.275,-68.755,44.816,156.8422,29.2978,0.0000
C00567=-46.575,-66.037,43.611,154.5478,28.5548,0.0000
C00568=-47.238,-63.546,42.745,151.9928,27.3092,0.0000
C00569=-49.870,-60.750,42.402,149.1164,25.1946,0.0000
C00570=-52.774,-58.195,42.387,148.7408,24.9413,0.0000
C00571=-55.552,-55.552,42.397,150.0514,26.5296,0.0000
C00572=-58.195,-52.774,42.387,151.4518,28.0677,0.0000
C00573=-60.750,-49.870,42.402,151.2690,27.6747,0.0000
C00574=-63.546,-47.238,42.745,149.6793,24.6603,0.0000
C00575=-66.037,-46.575,43.611,148.9232,22.1779,0.0000
C00576=-68.755,-47.275,44.816,148.6044,20.0576,0.0000
C00577=-71.950,-48.737,46.074,148.5724,17.5715,0.0000
C00578=-75.478,-50.465,47.055,149.0612,14.0880,0.0000
C00579=-79.009,-51.741,47.546,150.9695,8.7582,0.0000
C00580=-82.869,-51.201,47.807,157.9982,0.8532,0.0000
C00581=-86.517,-48.823,48.020,165.7127,-1.8078,0.0000
C00582=-89.240,-44.981,48.237,169.8709,-2.1105,0.0000
C00583=-91.399,-40.555,48.381,171.9062,-2.0151,0.0000
C00584=-93.306,-35.952,48.381,-172.8361,4.2800,0.0000
C00585=-94.909,-31.296,48.237,-171.3126,5.6373,0.0000
C00586=-95.700,-26.654,48.020,-168.5192,8.7492,0.0000
C00587=-94.802,-22.392,47.807,-164.6580,15.9863,0.0000
C00588=-92.454,-19.281,47.546,-165.0047,26.5387,0.0000
C00589=-89.056,-17.687,47.055,-167.7588,31.6493,0.0000
C00590=-85.339,-16.414,46.074,-170.3698,34.4000,0.0000
C00591=-82.045,-15.189,44.816,-172.6440,36.0530,0.0000
C00592=-79.628,-13.762,43.611,-174.8791,37.2229,0.0000
C00593=-78.336,-11.532,42.745,-177.8553,38.2761,0.0000
C00594=-78.220,-7.694,42.402,177.9782,39.0086,0.0000
C00595=-78.467,-3.833,42.387,177.4495,39.1155,0.0000
C00596=-78.562,0.000,42.397,-179.9998,39.1734,0.0000
C00597=-78.467,3.833,42.387,-177.4498,39.1155,0.0000
C00598=-78.220,7.694,42.402,-177.9795,39.0085,0.0000
C00599=-78.336,11.532,42.745,177.8547,38.2760,0.0000
C00600=-79.628,13.762,43.611,174.8791,37.2228,0.0000
C00601=-82.045,15.189,44.816,172.6443,36.0530,0.0000
C00602=-85.339,16.414,46.074,170.3703,34.4002,0.0000
C00603=-89.056,17.687,47.055,167.7593,31.6496,0.0000
C00604=-92.454,19.281,47.546,165.0050,26.5390,0.0000
C00605=-94.802,22.392,47.807,164.6580,15.9863,0.0000
C00606=-95.700,26.654,48.020,168.5192,8.7492,0.0000
C00607=-94.909,31.296,48.237,171.3126,5.6373,0.0000
C00608=-93.306,35.952,48.381,172.8361,4.2800,0.0000
C00609=-91.399,40.555,48.381,-171.9062,-2.0151,0.0000
C00610=-89.240,44.981,48.237,-169.8709,-2.1105,0.0000
C00611=-86.517,48.823,48.020,-165.7127,-1.8078,0.0000
C00612=-82.869,51.201,47.807,-157.9982,0.8532,0.0000
C00613=-79.009,51.741,47.546,-150.9696,8.7579,0.0000
C00614=-75.478,50.465,47.055,-149.0612,14.0876,0.0000
C00615=-71.950,48.737,46.074,-148.5722,17.5711,0.0000
C00616=-68.755,47.275,44.816,-148.6043,20.0574,0.0000
C00617=-66.037,46.575,43.611,-148.9231,22.1779,0.0000
C00618=-63.546,47.238,42.745,-149.6795,24.6607,0.0000
C00619=-60.750,49.870,42.402,-151.2696,27.6755,0.0000
C00620=-58.195,52.774,42.387,-151.4520,28.0679,0.0000
C00621=-55.552,55.552,42.397,-150.0512,26.5294,0.0000
C00622=-52.774,58.195,42.387,-148.7409,24.9415,0.0000
C00623=-49.870,60.750,42.402,-149.1172,25.1953,0.0000
C00624=-47.238,63.546,42.745,-151.9932,27.3095,0.0000
C00625=-46.575,66.037,43.611,-154.5477,28.5547,0.0000
C00626=-47.275,68.755,44.816,-156.8420,29.2977,0.0000
C00627=-48.737,71.950,46.074,-159.6394,29.8078,0.0000
C00628=-50.465,75.478,47.055,-163.6910,29.9113,0.0000
C00629=-51.741,79.009,47.546,-170.0072,28.6603,0.0000
C00630=-51.201,82.869,47.807,-179.0798,21.9992,0.0000
C00631=-48.823,86.517,48.020,178.1345,14.2800,0.0000
C00632=-44.981,89.240,48.237,177.8561,10.1221,0.0000
C00633=-40.555,91.399,48.381,177.9646,8.0888,0.0000
C00634=-35.952,93.306,48.381,-175.6864,-7.1438,0.0000
C00635=-31.296,94.909,48.237,-174.2977,-8.6450,0.0000
C00636=-26.654,95.700,48.020,-171.0751,-11.3454,0.0000
C00637=-22.392,94.802,47.807,-163.4548,-14.7350,0.0000
C00638=-19.281,92.454,47.546,-152.6593,-13.3838,0.0000
C00639=-17.687,89.056,47.055,-147.7588,-10.3981,0.0000
C00640=-16.414,85.339,46.074,-145.2198,-7.9336,0.0000
C00641=-15.189,82.045,44.816,-143.7214,-5.9412,0.0000
C00642=-13.762,79.628,43.611,-142.6667,-4.0757,0.0000
C00643=-11.532,78.336,42.745,-141.7045,-1.6840,0.0000
C00644=-7.694,78.220,42.402,-140.9740,1.5699,0.0000
C00645=-3.833,78.467,42.387,-140.8567,1.9784,0.0000
C00646=0.000,78.562,42.397,-140.8266,0.0001,0.0000
C00647=0.000,77.178,44.107,-140.7459,0.0001,0.0000
C00648=3.707,77.088,44.096,-140.7757,-1.9651,0.0000
C00649=7.481,76.852,44.112,-140.8928,-1.4913,0.0000
C00650=11.270,77.011,44.481,-141.6345,1.8462,0.0000
C00651=13.439,78.412,45.416,-142.5916,4.2404,0.0000
C00652=14.814,81.004,46.718,-143.6407,6.1180,0.0000
C00653=16.001,84.532,48.079,-145.1743,8.1791,0.0000
C00654=17.239,88.522,49.141,-147.8829,10.7909,0.0000
C00655=18.791,92.187,49.674,-153.4009,13.9431,0.0000
C00656=21.929,94.746,49.957,-165.5942,14.4192,0.0000
C00657=26.285,95.767,50.188,-172.9480,10.1040,0.0000
C00658=31.062,94.986,50.423,-175.6441,7.3403,0.0000
C00659=35.872,93.336,50.579,-176.7099,5.9809,0.0000
C00660=40.633,91.364,50.579,178.0782,-6.5482,0.0000
C00661=45.201,89.129,50.423,177.8530,-8.2566,0.0000
C00662=49.131,86.304,50.188,177.7384,-12.0941,0.0000
C00663=51.489,82.502,49.957,179.6518,-20.2709,0.0000
C00664=51.899,78.473,49.674,-171.0359,-28.5326,0.0000
C00665=50.405,74.784,49.141,-164.1063,-30.1109,0.0000
C00666=48.459,71.088,48.079,-159.7906,-30.0203,0.0000
C00667=46.803,67.754,46.718,-156.9050,-29.4839,0.0000
C00668=45.943,64.949,45.416,-154.6023,-28.7292,0.0000
C00669=46.486,62.424,44.481,-152.0458,-27.4798,0.0000
C00670=49.053,59.633,44.112,-149.0986,-25.3071,0.0000
C00671=51.888,57.130,44.096,-148.6786,-25.0010,0.0000
C00672=54.573,54.573,44.107,-149.9801,-26.5789,0.0000
C00673=57.130,51.888,44.096,-151.3704,-28.1076,0.0000
C00674=59.633,49.053,44.112,-151.1414,-27.6625,0.0000
C00675=62.424,46.486,44.482,-149.5093,-24.5741,0.0000
C00676=64.949,45.943,45.416,-148.7510,-22.0924,0.0000
C00677=67.754,46.803,46.718,-148.4226,-19.9659,0.0000
C00678=71.088,48.459,48.079,-148.3783,-17.4045,0.0000
C00679=74.784,50.405,49.141,-148.9107,-13.7041,0.0000
C00680=78.473,51.899,49.674,-151.1708,-7.8684,0.0000
C00681=82.502,51.489,49.957,-159.7288,0.3267,0.0000
C00682=86.304,49.131,50.188,-167.8968,2.2114,0.0000
C00683=89.129,45.201,50.423,-171.7377,2.1248,0.0000
C00684=91.364,40.633,50.579,-173.4481,1.9093,0.0000
C00685=93.336,35.872,50.579,174.0093,-3.2722,0.0000
C00686=94.986,31.062,50.423,172.6387,-4.3201,0.0000
C00687=95.767,26.285,50.188,169.8205,-6.9421,0.0000
C00688=94.746,21.929,49.957,165.1331,-13.9427,0.0000
C00689=92.187,18.791,49.674,164.4821,-25.7569,0.0000
C00690=88.522,17.239,49.141,167.3178,-31.4833,0.0000
C00691=84.532,16.001,48.079,170.0688,-34.4212,0.0000
C00692=81.004,14.814,46.718,172.4185,-36.1194,0.0000
C00693=78.412,13.439,45.416,174.6674,-37.2886,0.0000
C00694=77.011,11.270,44.481,177.6459,-38.3420,0.0000
C00695=76.852,7.481,44.112,-178.0784,-39.0914,0.0000
C00696=77.088,3.707,44.096,-177.4640,-39.1968,0.0000
C00697=77.178,0.000,44.107,179.9999,-39.2541,0.0000
C00698=77.088,-3.707,44.096,177.4641,-39.1969,0.0000
C00699=76.852,-7.481,44.112,178.0797,-39.0913,0.0000
C00700=77.011,-11.270,44.482,-177.6453,-38.3418,0.0000
C00701=78.412,-13.439,45.416,-174.6674,-37.2885,0.0000
C00702=81.004,-14.814,46.718,-172.4188,-36.1195,0.0000
C00703=84.532,-16.001,48.079,-170.0692,-34.4214,0.0000
C00704=88.522,-17.239,49.141,-167.3182,-31.4836,0.0000
C00705=92.187,-18.791,49.674,-164.4823,-25.7572,0.0000
C00706=94.746,-21.929,49.957,-165.1331,-13.9427,0.0000
C00707=95.767,-26.285,50.188,-169.8205,-6.9421,0.0000
C00708=94.986,-31.062,50.423,-172.6387,-4.3201,0.0000
C00709=93.336,-35.872,50.579,-174.0093,-3.2722,0.0000
C00710=91.364,-40.633,50.579,173.4481,1.9093,0.0000
C00711=89.129,-45.201,50.423,171.7377,2.1248,0.0000
C00712=86.304,-49.131,50.188,167.8968,2.2114,0.0000
C00713=82.502,-51.489,49.957,159.7288,0.3267,0.0000
C00714=78.473,-51.899,49.674,151.1709,-7.8680,0.0000
C00715=74.784,-50.405,49.141,148.9107,-13.7036,0.0000
C00716=71.088,-48.459,48.079,148.3782,-17.4041,0.0000
C00717=67.754,-46.803,46.718,148.4225,-19.9657,0.0000
C00718=64.949,-45.943,45.416,148.7510,-22.0925,0.0000
C00719=62.424,-46.486,44.481,149.5095,-24.5745,0.0000
C00720=59.633,-49.053,44.112,151.1420,-27.6633,0.0000
C00721=57.130,-51.888,44.096,151.3706,-28.1076,0.0000
C00722=54.573,-54.573,44.107,149.9800,-26.5788,0.0000
C00723=51.888,-57.130,44.096,148.6787,-25.0012,0.0000
C00724=49.053,-59.633,44.112,149.0994,-25.3078,0.0000
C00725=46.486,-62.424,44.482,152.0462,-27.4801,0.0000
C00726=45.943,-64.949,45.416,154.6023,-28.7292,0.0000
C00727=46.803,-67.754,46.718,156.9048,-29.4838,0.0000
C00728=48.459,-71.088,48.079,159.7902,-30.0201,0.0000
C00729=50.405,-74.784,49.141,164.1057,-30.1108,0.0000
C00730=51.899,-78.473,49.674,171.0355,-28.5327,0.0000
C00731=51.489,-82.502,49.957,-179.6518,-20.2709,0.0000
C00732=49.131,-86.304,50.188,-177.7384,-12.0941,0.0000
C00733=45.201,-89.129,50.423,-177.8530,-8.2566,0.0000
C00734=40.633,-91.364,50.579,-178.0782,-6.5482,0.0000
C00735=35.872,-93.336,50.579,176.7099,5.9809,0.0000
C00736=31.062,-94.986,50.423,175.6441,7.3403,0.0000
C00737=26.285,-95.767,50.188,172.9480,10.1040,0.0000
C00738=21.929,-94.746,49.957,165.5942,14.4192,0.0000
C00739=18.791,-92.187,49.674,153.4009,13.9431,0.0000
C00740=17.239,-88.522,49.141,147.8829,10.7909,0.0000
C00741=16.001,-84.532,48.079,145.1743,8.1791,0.0000
C00742=14.814,-81.004,46.718,143.6407,6.1180,0.0000
C00743=13.439,-78.412,45.416,142.5916,4.2404,0.0000
C00744=11.270,-77.011,44.481,141.6345,1.8462,0.0000
C00745=7.481,-76.852,44.112,140.8928,-1.4913,0.0000
C00746=3.707,-77.088,44.096,140.7757,-1.9651,0.0000
C00747=0.000,-77.178,44.107,140.7459,0.0001,0.0000
C00748=0.000,-77.178,44.107,140.7459,0.0001,0.0000
C00749=-3.707,-77.088,44.096,140.7756,1.9650,0.0000
C00750=-7.481,-76.852,44.112,140.8930,1.4903,0.0000
C00751=-11.270,-77.011,44.482,141.6346,-1.8466,0.0000
C00752=-13.439,-78.412,45.416,142.5916,-4.2404,0.0000
C00753=-14.814,-81.004,46.718,143.6407,-6.1178,0.0000
C00754=-16.001,-84.532,48.079,145.1742,-8.1787,0.0000
C00755=-17.239,-88.522,49.141,147.8826,-10.7905,0.0000
C00756=-18.791,-92.187,49.674,153.4006,-13.9429,0.0000
C00757=-21.929,-94.746,49.957,165.5942,-14.4192,0.0000
C00758=-26.285,-95.767,50.188,172.9480,-10.1040,0.0000
C00759=-31.062,-94.986,50.423,175.6441,-7.3403,0.0000
C00760=-35.872,-93.336,50.579,176.7099,-5.9809,0.0000
C00761=-40.633,-91.364,50.579,-178.0782,6.5482,0.0000
C00762=-45.201,-89.129,50.423,-177.8530,8.2566,0.0000
C00763=-49.131,-86.304,50.188,-177.7384,12.0941,0.0000
C00764=-51.489,-82.502,49.957,-179.6518,20.2709,0.0000
C00765=-51.899,-78.473,49.674,171.0359,28.5326,0.0000
C00766=-50.405,-74.784,49.141,164.1063,30.1109,0.0000
C00767=-48.459,-71.088,48.079,159.7906,30.0203,0.0000
C00768=-46.803,-67.754,46.718,156.9050,29.4839,0.0000
C00769=-45.943,-64.949,45.416,154.6023,28.7292,0.0000
C00770=-46.486,-62.424,44.481,152.0458,27.4798,0.0000
C00771=-49.053,-59.633,44.112,149.0986,25.3071,0.0000
C00772=-51.888,-57.130,44.096,148.6786,25.0010,0.0000
C00773=-54.573,-54.573,44.107,149.9801,26.5789,0.0000
C00774=-57.130,-51.888,44.096,151.3704,28.1076,0.0000
C00775=-59.633,-49.053,44.112,151.1414,27.6625,0.0000
C00776=-62.424,-46.486,44.482,149.5093,24.5741,0.0000
C00777=-64.949,-45.943,45.416,148.7510,22.0924,0.0000
C00778=-67.754,-46.803,46.718,148.4226,19.9659,0.0000
C00779=-71.088,-48.459,48.079,148.3783,17.4045,0.0000
C00780=-74.784,-50.405,49.141,148.9107,13.7041,0.0000
C00781=-78.473,-51.899,49.674,151.1708,7.8684,0.0000
C00782=-82.502,-51.489,49.957,159.7288,-0.3267,0.0000
C00783=-86.304,-49.131,50.188,167.8968,-2.2114,0.0000
C00784=-89.129,-45.201,50.423,171.7377,-2.1248,0.0000
C00785=-91.364,-40.633,50.579,173.4481,-1.9093,0.0000
C00786=-93.336,-35.872,50.579,-174.0093,3.2722,0.0000
C00787=-94.986,-31.062,50.423,-172.6387,4.3201,0.0000
C00788=-95.767,-26.285,50.188,-169.8205,6.9421,0.0000
C00789=-94.746,-21.929,49.957,-165.1331,13.9427,0.0000
C00790=-92.187,-18.791,49.674,-164.4821,25.7569,0.0000
C00791=-88.522,-17.239,49.141,-167.3178,31.4833,0.0000
C00792=-84.532,-16.001,48.079,-170.0688,34.4212,0.0000
C00793=-81.004,-14.814,46.718,-172.4185,36.1194,0.0000
C00794=-78.412,-13.439,45.416,-174.6674,37.2886,0.0000
C00795=-77.011,-11.270,44.481,-177.6459,38.3420,0.0000
C00796=-76.852,-7.481,44.112,178.0784,39.0914,0.0000
C00797=-77.088,-3.707,44.096,177.4640,39.1968,0.0000
C00798=-77.178,0.000,44.107,-179.9999,39.2541,0.0000
C00799=-77.088,3.707,44.096,-177.4641,39.1969,0.0000
C00800=-76.852,7.481,44.112,-178.0797,39.0913,0.0000
C00801=-77.011,11.270,44.482,177.6453,38.3418,0.0000
C00802=-78.412,13.439,45.416,174.6674,37.2885,0.0000
C00803=-81.004,14.814,46.718,172.4188,36.1195,0.0000
C00804=-84.532,16.001,48.079,170.0692,34.4214,0.0000
C00805=-88.522,17.239,49.141,167.3182,31.4836,0.0000
C00806=-92.187,18.791,49.674,164.4823,25.7572,0.0000
C00807=-94.746,21.929,49.957,165.1331,13.9427,0.0000
C00808=-95.767,26.285,50.188,169.8205,6.9421,0.0000
C00809=-94.986,31.062,50.423,172.6387,4.3201,0.0000
C00810=-93.336,35.872,50.579,174.0093,3.2722,0.0000
C00811=-91.364,40.633,50.579,-173.4481,-1.9093,0.0000
C00812=-89.129,45.201,50.423,-171.7377,-2.1248,0.0000
C00813=-86.304,49.131,50.188,-167.8968,-2.2114,0.0000
C00814=-82.502,51.489,49.957,-159.7288,-0.3267,0.0000
C00815=-78.473,51.899,49.674,-151.1709,7.8680,0.0000
C00816=-74.784,50.405,49.141,-148.9107,13.7036,0.0000
C00817=-71.088,48.459,48.079,-148.3782,17.4041,0.0000
C00818=-67.754,46.803,46.718,-148.4225,19.9657,0.0000
C00819=-64.949,45.943,45.416,-148.7510,22.0925,0.0000
C00820=-62.424,46.486,44.481,-149.5095,24.5745,0.0000
C00821=-59.633,49.053,44.112,-151.1420,27.6633,0.0000
C00822=-57.130,51.888,44.096,-151.3706,28.1076,0.0000
C00823=-54.573,54.573,44.107,-149.9800,26.5788,0.0000
C00824=-51.888,57.130,44.096,-148.6787,25.0012,0.0000
C00825=-49.053,59.633,44.112,-149.0994,25.3078,0.0000
C00826=-46.486,62.424,44.482,-152.0462,27.4801,0.0000
C00827=-45.943,64.949,45.416,-154.6023,28.7292,0.0000
C00828=-46.803,67.754,46.718,-156.9048,29.4838,0.0000
C00829=-48.459,71.088,48.079,-159.7902,30.0201,0.0000
C00830=-50.405,74.784,49.141,-164.1057,30.1108,0.0000
C00831=-51.899,78.473,49.674,-171.0355,28.5327,0.0000
C00832=-51.489,82.502,49.957,179.6518,20.2709,0.0000
C00833=-49.131,86.304,50.188,177.7384,12.0941,0.0000
C00834=-45.201,89.129,50.423,177.8530,8.2566,0.0000
C00835=-40.633,91.364,50.579,178.0782,6.5482,0.0000
C00836=-35.872,93.336,50.579,-176.7099,-5.9809,0.0000
C00837=-31.062,94.986,50.423,-175.6441,-7.3403,0.0000
C00838=-26.285,95.767,50.188,-172.9480,-10.1040,0.0000
C00839=-21.929,94.746,49.957,-165.5942,-14.4192,0.0000
C00840=-18.791,92.187,49.674,-153.4006,-13.9429,0.0000
C00841=-17.239,88.522,49.141,-147.8826,-10.7905,0.0000
C00842=-16.001,84.532,48.079,-145.1742,-8.1787,0.0000
C00843=-14.814,81.004,46.718,-143.6407,-6.1178,0.0000
C00844=-13.439,78.412,45.416,-142.5916,-4.2404,0.0000
C00845=-11.270,77.011,44.482,-141.6346,-1.8466,0.0000
C00846=-7.481,76.852,44.112,-140.8930,1.4903,0.0000
C00847=-3.707,77.088,44.096,-140.7756,1.9650,0.0000
C00848=0.000,77.178,44.107,-140.7459,0.0001,0.0000
C00849=0.000,75.789,45.812,-140.7136,0.0000,0.0000
C00850=3.580,75.703,45.801,-140.7430,-1.9483,0.0000
C00851=7.267,75.480,45.818,-140.8601,-1.4151,0.0000
C00852=11.008,75.681,46.215,-141.6117,1.9948,0.0000
C00853=13.116,77.193,47.218,-142.5616,4.3856,0.0000
C00854=14.439,79.961,48.618,-143.6041,6.2745,0.0000
C00855=15.588,83.726,50.084,-145.1762,8.4096,0.0000
C00856=16.791,87.989,51.229,-148.0851,11.1872,0.0000
C00857=18.302,91.921,51.802,-154.3991,14.5035,0.0000
C00858=21.467,94.690,52.107,-168.0122,13.6646,0.0000
C00859=25.919,95.834,52.356,-174.7421,8.5379,0.0000
C00860=30.830,95.062,52.610,-176.8657,5.8797,0.0000
C00861=35.794,93.367,52.777,-177.6296,4.7306,0.0000
C00862=40.710,91.330,52.777,178.3220,-5.0175,0.0000
C00863=45.419,89.019,52.610,178.0408,-6.3669,0.0000
C00864=49.437,86.092,52.356,177.6217,-9.7332,0.0000
C00865=51.776,82.136,52.107,178.5335,-18.0446,0.0000
C00866=52.057,77.939,51.802,-172.2568,-28.2221,0.0000
C00867=50.345,74.091,51.229,-164.5897,-30.2587,0.0000
C00868=48.181,70.226,50.084,-159.9709,-30.1900,0.0000
C00869=46.331,66.751,48.618,-156.9911,-29.6261,0.0000
C00870=45.309,63.858,47.218,-154.6823,-28.8598,0.0000
C00871=45.731,61.299,46.215,-152.1306,-27.6101,0.0000
C00872=48.234,58.511,45.818,-149.1210,-25.3875,0.0000
C00873=50.999,56.061,45.801,-148.6611,-25.0341,0.0000
C00874=53.591,53.591,45.812,-149.9515,-26.5986,0.0000
C00875=56.061,50.999,45.801,-151.3296,-28.1147,0.0000
C00876=58.511,48.233,45.818,-151.0591,-27.6229,0.0000
C00877=61.299,45.731,46.215,-149.3899,-24.4701,0.0000
C00878=63.858,45.309,47.218,-148.6304,-21.9949,0.0000
C00879=66.751,46.331,48.618,-148.2909,-19.8633,0.0000
C00880=70.226,48.181,50.084,-148.2330,-17.2204,0.0000
C00881=74.091,50.345,51.229,-148.8201,-13.2697,0.0000
C00882=77.939,52.057,51.802,-151.5585,-6.8184,0.0000
C00883=82.136,51.776,52.107,-161.9499,1.3943,0.0000
C00884=86.092,49.437,52.356,-170.2586,2.3440,0.0000
C00885=89.019,45.419,52.610,-173.6294,1.9471,0.0000
C00886=91.330,40.710,52.777,-174.9803,1.6715,0.0000
C00887=93.367,35.794,52.777,175.2654,-2.3623,0.0000
C00888=95.062,30.830,52.610,174.1115,-3.1178,0.0000
C00889=95.834,25.919,52.356,171.4265,-5.1995,0.0000
C00890=94.690,21.467,52.107,166.0426,-11.6437,0.0000
C00891=91.921,18.302,51.802,163.9948,-24.7292,0.0000
C00892=87.989,16.791,51.229,166.8844,-31.2393,0.0000
C00893=83.726,15.588,50.084,169.7910,-34.3964,0.0000
C00894=79.961,14.439,48.618,172.2217,-36.1433,0.0000
C00895=77.193,13.116,47.218,174.4829,-37.3100,0.0000
C00896=75.681,11.008,46.215,177.4556,-38.3608,0.0000
C00897=75.480,7.267,45.818,-178.1757,-39.1257,0.0000
C00898=75.703,3.580,45.801,-177.4844,-39.2300,0.0000
C00899=75.789,0.000,45.812,180.0000,-39.2864,0.0000
C00900=75.703,-3.580,45.801,177.4845,-39.2300,0.0000
C00901=75.480,-7.267,45.818,178.1770,-39.1256,0.0000
C00902=75.681,-11.008,46.215,-177.4551,-38.3606,0.0000
C00903=77.193,-13.116,47.218,-174.4829,-37.3100,0.0000
C00904=79.961,-14.439,48.618,-172.2220,-36.1434,0.0000
C00905=83.726,-15.588,50.084,-169.7914,-34.3966,0.0000
C00906=87.989,-16.791,51.229,-166.8848,-31.2397,0.0000
C00907=91.921,-18.302,51.802,-163.9950,-24.7295,0.0000
C00908=94.690,-21.467,52.107,-166.0426,-11.6437,0.0000
C00909=95.834,-25.919,52.356,-171.4265,-5.1995,0.0000
C00910=95.062,-30.830,52.610,-174.1115,-3.1178,0.0000
C00911=93.367,-35.794,52.777,-175.2654,-2.3623,0.0000
C00912=91.330,-40.710,52.777,174.9803,1.6715,0.0000
C00913=89.019,-45.419,52.610,173.6294,1.9471,0.0000
C00914=86.092,-49.437,52.356,170.2586,2.3440,0.0000
C00915=82.136,-51.776,52.107,161.9499,1.3943,0.0000
C00916=77.939,-52.057,51.802,151.5586,-6.8180,0.0000
C00917=74.091,-50.345,51.229,148.8201,-13.2691,0.0000
C00918=70.226,-48.181,50.084,148.2329,-17.2200,0.0000
C00919=66.751,-46.331,48.618,148.2908,-19.8632,0.0000
C00920=63.858,-45.309,47.218,148.6304,-21.9950,0.0000
C00921=61.299,-45.731,46.215,149.3901,-24.4705,0.0000
C00922=58.511,-48.234,45.818,151.0597,-27.6238,0.0000
C00923=56.061,-50.999,45.801,151.3297,-28.1148,0.0000
C00924=53.591,-53.591,45.812,149.9515,-26.5986,0.0000
C00925=50.999,-56.061,45.801,148.6611,-25.0342,0.0000
C00926=48.233,-58.511,45.818,149.1218,-25.3883,0.0000
C00927=45.731,-61.299,46.215,152.1310,-27.6104,0.0000
C00928=45.309,-63.858,47.218,154.6824,-28.8598,0.0000
C00929=46.331,-66.751,48.618,156.9909,-29.6260,0.0000
C00930=48.181,-70.226,50.084,159.9705,-30.1898,0.0000
C00931=50.345,-74.091,51.229,164.5892,-30.2586,0.0000
C00932=52.057,-77.939,51.802,172.2564,-28.2222,0.0000
C00933=51.776,-82.136,52.107,-178.5335,-18.0446,0.0000
C00934=49.437,-86.092,52.356,-177.6217,-9.7332,0.0000
C00935=45.419,-89.019,52.610,-178.0408,-6.3669,0.0000
C00936=40.710,-91.330,52.777,-178.3220,-5.0175,0.0000
C00937=35.794,-93.367,52.777,177.6296,4.7306,0.0000
C00938=30.830,-95.062,52.610,176.8657,5.8797,0.0000
C00939=25.919,-95.834,52.356,174.7421,8.5379,0.0000
C00940=21.467,-94.690,52.107,168.0122,13.6646,0.0000
C00941=18.302,-91.921,51.802,154.3991,14.5035,0.0000
C00942=16.791,-87.989,51.229,148.0851,11.1872,0.0000
C00943=15.588,-83.726,50.084,145.1762,8.4096,0.0000
C00944=14.439,-79.961,48.618,143.6041,6.2745,0.0000
C00945=13.116,-77.193,47.218,142.5616,4.3856,0.0000
C00946=11.008,-75.681,46.215,141.6117,1.9948,0.0000
C00947=7.267,-75.480,45.818,140.8601,-1.4151,0.0000
C00948=3.580,-75.703,45.801,140.7430,-1.9483,0.0000
C00949=0.000,-75.789,45.812,140.7136,0.0000,0.0000
C00950=0.000,-75.789,45.812,140.7136,0.0000,0.0000
C00951=-3.580,-75.703,45.801,140.7429,1.9483,0.0000
C00952=-7.267,-75.480,45.818,140.8602,1.4141,0.0000
C00953=-11.008,-75.681,46.215,141.6118,-1.9953,0.0000
C00954=-13.116,-77.193,47.218,142.5617,-4.3856,0.0000
C00955=-14.439,-79.961,48.618,143.6040,-6.2744,0.0000
C00956=-15.588,-83.726,50.084,145.1760,-8.4092,0.0000
C00957=-16.791,-87.989,51.229,148.0848,-11.1868,0.0000
C00958=-18.302,-91.921,51.802,154.3988,-14.5033,0.0000
C00959=-21.467,-94.690,52.107,168.0122,-13.6646,0.0000
C00960=-25.919,-95.834,52.356,174.7421,-8.5379,0.0000
C00961=-30.830,-95.062,52.610,176.8657,-5.8797,0.0000
C00962=-35.794,-93.367,52.777,177.6296,-4.7306,0.0000
C00963=-40.710,-91.330,52.777,-178.3220,5.0175,0.0000
C00964=-45.419,-89.019,52.610,-178.0408,6.3669,0.0000
C00965=-49.437,-86.092,52.356,-177.6217,9.7332,0.0000
C00966=-51.776,-82.136,52.107,-178.5335,18.0446,0.0000
C00967=-52.057,-77.939,51.802,172.2568,28.2221,0.0000
C00968=-50.345,-74.091,51.229,164.5897,30.2587,0.0000
C00969=-48.181,-70.226,50.084,159.9709,30.1900,0.0000
C00970=-46.331,-66.751,48.618,156.9911,29.6261,0.0000
C00971=-45.309,-63.858,47.218,154.6823,28.8598,0.0000
C00972=-45.731,-61.299,46.215,152.1306,27.6101,0.0000
C00973=-48.234,-58.511,45.818,149.1210,25.3875,0.0000
C00974=-50.999,-56.061,45.801,148.6611,25.0341,0.0000
C00975=-53.591,-53.591,45.812,149.9515,26.5986,0.0000
C00976=-56.061,-50.999,45.801,151.3296,28.1147,0.0000
C00977=-58.511,-48.233,45.818,151.0591,27.6229,0.0000
C00978=-61.299,-45.731,46.215,149.3899,24.4701,0.0000
C00979=-63.858,-45.309,47.218,148.6304,21.9949,0.0000
C00980=-66.751,-46.331,48.618,148.2909,19.8633,0.0000
C00981=-70.226,-48.181,50.084,148.2330,17.2204,0.0000
C00982=-74.091,-50.345,51.229,148.8201,13.2697,0.0000
C00983=-77.939,-52.057,51.802,151.5585,6.8184,0.0000
C00984=-82.136,-51.776,52.107,161.9499,-1.3943,0.0000
C00985=-86.092,-49.437,52.356,170.2586,-2.3440,0.0000
C00986=-89.019,-45.419,52.610,173.6294,-1.9471,0.0000
C00987=-91.330,-40.710,52.777,174.9803,-1.6715,0.0000
C00988=-93.367,-35.794,52.777,-175.2654,2.3623,0.0000
C00989=-95.062,-30.830,52.610,-174.1115,3.1178,0.0000
C00990=-95.834,-25.919,52.356,-171.4265,5.1995,0.0000
C00991=-94.690,-21.467,52.107,-166.0426,11.6437,0.0000
C00992=-91.921,-18.302,51.802,-163.9948,24.7292,0.0000
C00993=-87.989,-16.791,51.229,-166.8844,31.2393,0.0000
C00994=-83.726,-15.588,50.084,-169.7910,34.3964,0.0000
C00995=-79.961,-14.439,48.618,-172.2217,36.1433,0.0000
C00996=-77.193,-13.116,47.218,-174.4829,37.3100,0.0000
C00997=-75.681,-11.008,46.215,-177.4556,38.3608,0.0000
C00998=-75.480,-7.267,45.818,178.1757,39.1257,0.0000
C00999=-75.703,-3.580,45.801,177.4844,39.2300,0.0000
C01000=-75.789,0.000,45.812,-180.0000,39.2864,0.0000
C01001=-75.703,3.580,45.801,-177.4845,39.2300,0.0000
C01002=-75.480,7.267,45.818,-178.1770,39.1256,0.0000
C01003=-75.681,11.008,46.215,177.4551,38.3606,0.0000
C01004=-77.193,13.116,47.218,174.4829,37.3100,0.0000
C01005=-79.961,14.439,48.618,172.2220,36.1434,0.0000
C01006=-83.726,15.588,50.084,169.7914,34.3966,0.0000
C01007=-87.989,16.791,51.229,166.8848,31.2397,0.0000
C01008=-91.921,18.302,51.802,163.9950,24.7295,0.0000
C01009=-94.690,21.467,52.107,166.0426,11.6437,0.0000
C01010=-95.834,25.919,52.356,171.4265,5.1995,0.0000
C01011=-95.062,30.830,52.610,174.1115,3.1178,0.0000
C01012=-93.367,35.794,52.777,175.2654,2.3623,0.0000
C01013=-91.330,40.710,52.777,-174.9803,-1.6715,0.0000
C01014=-89.019,45.419,52.610,-173.6294,-1.9471,0.0000
C01015=-86.092,49.437,52.356,-170.2586,-2.3440,0.0000
C01016=-82.136,51.776,52.107,-161.9499,-1.3943,0.0000
C01017=-77.939,52.057,51.802,-151.5586,6.8180,0.0000
C01018=-74.091,50.345,51.229,-148.8201,13.2691,0.0000
C01019=-70.226,48.181,50.084,-148.2329,17.2200,0.0000
C01020=-66.751,46.331,48.618,-148.2908,19.8632,0.0000
C01021=-63.858,45.309,47.218,-148.6304,21.9950,0.0000
C01022=-61.299,45.731,46.215,-149.3901,24.4705,0.0000
C01023=-58.511,48.234,45.818,-151.0597,27.6238,0.0000
C01024=-56.061,50.999,45.801,-151.3297,28.1148,0.0000
C01025=-53.591,53.591,45.812,-149.9515,26.5986,0.0000
C01026=-50.999,56.061,45.801,-148.6611,25.0342,0.0000
C01027=-48.233,58.511,45.818,-149.1218,25.3883,0.0000
C01028=-45.731,61.299,46.215,-152.1310,27.6104,0.0000
C01029=-45.309,63.858,47.218,-154.6824,28.8598,0.0000
C01030=-46.331,66.751,48.618,-156.9909,29.6260,0.0000
C01031=-48.181,70.226,50.084,-159.9705,30.1898,0.0000
C01032=-50.345,74.091,51.229,-164.5892,30.2586,0.0000
C01033=-52.057,77.939,51.802,-172.2564,28.2222,0.0000
C01034=-51.776,82.136,52.107,178.5335,18.0446,0.0000
C01035=-49.437,86.092,52.356,177.6217,9.7332,0.0000
C01036=-45.419,89.019,52.610,178.0408,6.3669,0.0000
C01037=-40.710,91.330,52.777,178.3220,5.0175,0.0000
C01038=-35.794,93.367,52.777,-177.6296,-4.7306,0.0000
C01039=-30.830,95.062,52.610,-176.8657,-5.8797,0.0000
C01040=-25.919,95.834,52.356,-174.7421,-8.5379,0.0000
C01041=-21.467,94.690,52.107,-168.0122,-13.6646,0.0000
C01042=-18.302,91.921,51.802,-154.3988,-14.5033,0.0000
C01043=-16.791,87.989,51.229,-148.0848,-11.1868,0.0000
C01044=-15.588,83.726,50.084,-145.1760,-8.4092,0.0000
C01045=-14.439,79.961,48.618,-143.6040,-6.2744,0.0000
C01046=-13.116,77.193,47.218,-142.5617,-4.3856,0.0000
C01047=-11.008,75.681,46.215,-141.6118,-1.9953,0.0000
C01048=-7.267,75.480,45.818,-140.8602,1.4141,0.0000
C01049=-3.580,75.703,45.801,-140.7429,1.9483,0.0000
C01050=0.000,75.789,45.812,-140.7136,0.0000,0.0000
C01051=0.000,74.396,47.516,-140.7285,-0.0001,0.0000
C01052=3.453,74.315,47.503,-140.7573,-1.9283,0.0000
C01053=7.053,74.105,47.522,-140.8742,-1.3427,0.0000
C01054=10.745,74.349,47.946,-141.6345,2.1294,0.0000
C01055=12.792,75.972,49.019,-142.5753,4.5119,0.0000
C01056=14.064,78.919,50.519,-143.6103,6.4123,0.0000
C01057=15.177,82.922,52.090,-145.2255,8.6279,0.0000
C01058=16.346,87.459,53.317,-148.3753,11.5930,0.0000
C01059=17.816,91.657,53.931,-155.7440,15.0466,0.0000
C01060=21.009,94.635,54.258,-170.6048,12.3676,0.0000
C01061=25.555,95.900,54.525,-176.3598,6.7215,0.0000
C01062=30.600,95.138,54.796,-177.9269,4.3294,0.0000
C01063=35.715,93.397,54.976,-178.4311,3.4353,0.0000
C01064=40.787,91.296,54.976,178.6769,-3.5372,0.0000
C01065=45.636,88.910,54.796,178.3978,-4.5245,0.0000
C01066=49.741,85.881,54.525,177.7942,-7.3164,0.0000
C01067=52.061,81.773,54.258,177.7005,-15.3195,0.0000
C01068=52.213,77.409,53.931,-173.7155,-27.6519,0.0000
C01069=50.285,73.401,53.317,-165.1535,-30.3519,0.0000
C01070=47.903,69.367,52.090,-160.1826,-30.3188,0.0000
C01071=45.859,65.749,50.519,-157.1004,-29.7261,0.0000
C01072=44.675,62.766,49.019,-154.7868,-28.9480,0.0000
C01073=44.975,60.171,47.946,-152.2457,-27.7008,0.0000
C01074=47.412,57.387,47.522,-149.1821,-25.4365,0.0000
C01075=50.108,54.990,47.503,-148.6870,-25.0414,0.0000
C01076=52.606,52.606,47.516,-149.9646,-26.5895,0.0000
C01077=54.990,50.108,47.503,-151.3283,-28.0902,0.0000
C01078=57.387,47.412,47.522,-151.0211,-27.5573,0.0000
C01079=60.171,44.975,47.946,-149.3197,-24.3495,0.0000
C01080=62.766,44.675,49.019,-148.5597,-21.8862,0.0000
C01081=65.749,45.859,50.519,-148.2076,-19.7499,0.0000
C01082=69.367,47.903,52.090,-148.1348,-17.0173,0.0000
C01083=73.401,50.285,53.317,-148.7928,-12.7748,0.0000
C01084=77.409,52.213,53.931,-152.2057,-5.5647,0.0000
C01085=81.773,52.061,54.258,-164.6687,2.2178,0.0000
C01086=85.881,49.741,54.525,-172.6782,2.1879,0.0000
C01087=88.910,45.636,54.796,-175.4737,1.5972,0.0000
C01088=91.296,40.787,54.976,-176.4619,1.3206,0.0000
C01089=93.397,35.715,54.976,176.5634,-1.5661,0.0000
C01090=95.138,30.600,54.796,175.6678,-2.0672,0.0000
C01091=95.900,25.555,54.525,173.2650,-3.6152,0.0000
C01092=94.635,21.009,54.258,167.4696,-9.1753,0.0000
C01093=91.657,17.816,53.931,163.5718,-23.3739,0.0000
C01094=87.459,16.346,53.317,166.4544,-30.9077,0.0000
C01095=82.922,15.177,52.090,169.5340,-34.3255,0.0000
C01096=78.919,14.064,50.519,172.0524,-36.1259,0.0000
C01097=75.972,12.792,49.019,174.3255,-37.2889,0.0000
C01098=74.349,10.745,47.946,177.2849,-38.3342,0.0000
C01099=74.105,7.053,47.522,-178.2694,-39.1130,0.0000
C01100=74.315,3.453,47.503,-177.5108,-39.2162,0.0000
C01101=74.396,0.000,47.516,-179.9999,-39.2715,0.0000
C01102=74.315,-3.453,47.503,177.5108,-39.2163,0.0000
C01103=74.105,-7.053,47.522,178.2707,-39.1129,0.0000
C01104=74.349,-10.745,47.946,-177.2844,-38.3341,0.0000
C01105=75.972,-12.792,49.019,-174.3254,-37.2889,0.0000
C01106=78.919,-14.064,50.519,-172.0526,-36.1260,0.0000
C01107=82.922,-15.177,52.090,-169.5344,-34.3256,0.0000
C01108=87.459,-16.346,53.317,-166.4548,-30.9081,0.0000
C01109=91.657,-17.816,53.931,-163.5720,-23.3743,0.0000
C01110=94.635,-21.009,54.258,-167.4696,-9.1753,0.0000
C01111=95.900,-25.555,54.525,-173.2650,-3.6152,0.0000
C01112=95.138,-30.600,54.796,-175.6678,-2.0672,0.0000
C01113=93.397,-35.715,54.976,-176.5634,-1.5661,0.0000
C01114=91.296,-40.787,54.976,176.4619,1.3206,0.0000
C01115=88.910,-45.636,54.796,175.4737,1.5972,0.0000
C01116=85.881,-49.741,54.525,172.6782,2.1879,0.0000
C01117=81.773,-52.061,54.258,164.6687,2.2178,0.0000
C01118=77.409,-52.213,53.931,152.2059,-5.5643,0.0000
C01119=73.401,-50.285,53.317,148.7928,-12.7743,0.0000
C01120=69.367,-47.903,52.090,148.1347,-17.0170,0.0000
C01121=65.749,-45.859,50.519,148.2075,-19.7497,0.0000
C01122=62.766,-44.675,49.019,148.5597,-21.8862,0.0000
C01123=60.171,-44.975,47.946,149.3199,-24.3499,0.0000
C01124=57.387,-47.412,47.522,151.0217,-27.5582,0.0000
C01125=54.990,-50.108,47.503,151.3284,-28.0902,0.0000
C01126=52.606,-52.606,47.516,149.9647,-26.5896,0.0000
C01127=50.108,-54.990,47.503,148.6870,-25.0415,0.0000
C01128=47.412,-57.387,47.522,149.1829,-25.4372,0.0000
C01129=44.975,-60.171,47.946,152.2461,-27.7011,0.0000
C01130=44.675,-62.766,49.019,154.7869,-28.9480,0.0000
C01131=45.859,-65.749,50.519,157.1002,-29.7260,0.0000
C01132=47.903,-69.367,52.090,160.1822,-30.3186,0.0000
C01133=50.285,-73.401,53.317,165.1529,-30.3518,0.0000
C01134=52.213,-77.409,53.931,173.7151,-27.6520,0.0000
C01135=52.061,-81.773,54.258,-177.7005,-15.3195,0.0000
C01136=49.741,-85.881,54.525,-177.7942,-7.3164,0.0000
C01137=45.636,-88.910,54.796,-178.3978,-4.5245,0.0000
C01138=40.787,-91.296,54.976,-178.6769,-3.5372,0.0000
C01139=35.715,-93.397,54.976,178.4311,3.4353,0.0000
C01140=30.600,-95.138,54.796,177.9269,4.3294,0.0000
C01141=25.555,-95.900,54.525,176.3598,6.7215,0.0000
C01142=21.009,-94.635,54.258,170.6048,12.3676,0.0000
C01143=17.816,-91.657,53.931,155.7440,15.0466,0.0000
C01144=16.346,-87.459,53.317,148.3753,11.5930,0.0000
C01145=15.177,-82.922,52.090,145.2255,8.6279,0.0000
C01146=14.064,-78.919,50.519,143.6103,6.4123,0.0000
C01147=12.792,-75.972,49.019,142.5753,4.5119,0.0000
C01148=10.745,-74.349,47.946,141.6345,2.1294,0.0000
C01149=7.053,-74.105,47.522,140.8742,-1.3427,0.0000
C01150=3.453,-74.315,47.503,140.7573,-1.9283,0.0000
C01151=0.000,-74.396,47.516,140.7285,-0.0001,0.0000
C01152=0.000,-74.396,47.516,140.7285,-0.0001,0.0000
C01153=-3.453,-74.315,47.503,140.7572,1.9283,0.0000
C01154=-7.053,-74.105,47.522,140.8743,1.3417,0.0000
C01155=-10.745,-74.349,47.946,141.6346,-2.1298,0.0000
C01156=-12.792,-75.972,49.019,142.5753,-4.5119,0.0000
C01157=-14.064,-78.919,50.519,143.6103,-6.4121,0.0000
C01158=-15.177,-82.922,52.090,145.2254,-8.6275,0.0000
C01159=-16.346,-87.459,53.317,148.3749,-11.5926,0.0000
C01160=-17.816,-91.657,53.931,155.7436,-15.0464,0.0000
C01161=-21.009,-94.635,54.258,170.6048,-12.3676,0.0000
C01162=-25.555,-95.900,54.525,176.3598,-6.7215,0.0000
C01163=-30.600,-95.138,54.796,177.9269,-4.3294,0.0000
C01164=-35.715,-93.397,54.976,178.4311,-3.4353,0.0000
C01165=-40.787,-91.296,54.976,-178.6769,3.5372,0.0000
C01166=-45.636,-88.910,54.796,-178.3978,4.5245,0.0000
C01167=-49.741,-85.881,54.525,-177.7942,7.3164,0.0000
C01168=-52.061,-81.773,54.258,-177.7005,15.3195,0.0000
C01169=-52.213,-77.409,53.931,173.7155,27.6519,0.0000
C01170=-50.285,-73.401,53.317,165.1535,30.3519,0.0000
C01171=-47.903,-69.367,52.090,160.1826,30.3188,0.0000
C01172=-45.859,-65.749,50.519,157.1004,29.7261,0.0000
C01173=-44.675,-62.766,49.019,154.7868,28.9480,0.0000
C01174=-44.975,-60.171,47.946,152.2457,27.7008,0.0000
C01175=-47.412,-57.387,47.522,149.1821,25.4365,0.0000
C01176=-50.108,-54.990,47.503,148.6870,25.0414,0.0000
C01177=-52.606,-52.606,47.516,149.9646,26.5895,0.0000
C01178=-54.990,-50.108,47.503,151.3283,28.0902,0.0000
C01179=-57.387,-47.412,47.522,151.0211,27.5573,0.0000
C01180=-60.171,-44.975,47.946,149.3197,24.3495,0.0000
C01181=-62.766,-44.675,49.019,148.5597,21.8862,0.0000
C01182=-65.749,-45.859,50.519,148.2076,19.7499,0.0000
C01183=-69.367,-47.903,52.090,148.1348,17.0173,0.0000
C01184=-73.401,-50.285,53.317,148.7928,12.7748,0.0000
C01185=-77.409,-52.213,53.931,152.2057,5.5647,0.0000
C01186=-81.773,-52.061,54.258,164.6687,-2.2178,0.0000
C01187=-85.881,-49.741,54.525,172.6782,-2.1879,0.0000
C01188=-88.910,-45.636,54.796,175.4737,-1.5972,0.0000
C01189=-91.296,-40.787,54.976,176.4619,-1.3206,0.0000
C01190=-93.397,-35.715,54.976,-176.5634,1.5661,0.0000
C01191=-95.138,-30.600,54.796,-175.6678,2.0672,0.0000
C01192=-95.900,-25.555,54.525,-173.2650,3.6152,0.0000
C01193=-94.635,-21.009,54.258,-167.4696,9.1753,0.0000
C01194=-91.657,-17.816,53.931,-163.5718,23.3739,0.0000
C01195=-87.459,-16.346,53.317,-166.4544,30.9077,0.0000
C01196=-82.922,-15.177,52.090,-169.5340,34.3255,0.0000
C01197=-78.919,-14.064,50.519,-172.0524,36.1259,0.0000
C01198=-75.972,-12.792,49.019,-174.3255,37.2889,0.0000
C01199=-74.349,-10.745,47.946,-177.2849,38.3342,0.0000
C01200=-74.105,-7.053,47.522,178.2694,39.1130,0.0000
C01201=-74.315,-3.453,47.503,177.5108,39.2162,0.0000
C01202=-74.396,0.000,47.516,179.9999,39.2715,0.0000
C01203=-74.315,3.453,47.503,-177.5108,39.2163,0.0000
C01204=-74.105,7.053,47.522,-178.2707,39.1129,0.0000
C01205=-74.349,10.745,47.946,177.2844,38.3341,0.0000
C01206=-75.972,12.792,49.019,174.3254,37.2889,0.0000
C01207=-78.919,14.064,50.519,172.0526,36.1260,0.0000
C01208=-82.922,15.177,52.090,169.5344,34.3256,0.0000
C01209=-87.459,16.346,53.317,166.4548,30.9081,0.0000
C01210=-91.657,17.816,53.931,163.5720,23.3743,0.0000
C01211=-94.635,21.009,54.258,167.4696,9.1753,0.0000
C01212=-95.900,25.555,54.525,173.2650,3.6152,0.0000
C01213=-95.138,30.600,54.796,175.6678,2.0672,0.0000
C01214=-93.397,35.715,54.976,176.5634,1.5661,0.0000
C01215=-91.296,40.787,54.976,-176.4619,-1.3206,0.0000
C01216=-88.910,45.636,54.796,-175.4737,-1.5972,0.0000
C01217=-85.881,49.741,54.525,-172.6782,-2.1879,0.0000
C01218=-81.773,52.061,54.258,-164.6687,-2.2178,0.0000
C01219=-77.409,52.213,53.931,-152.2059,5.5643,0.0000
C01220=-73.401,50.285,53.317,-148.7928,12.7743,0.0000
C01221=-69.367,47.903,52.090,-148.1347,17.0170,0.0000
C01222=-65.749,45.859,50.519,-148.2075,19.7497,0.0000
C01223=-62.766,44.675,49.019,-148.5597,21.8862,0.0000
C01224=-60.171,44.975,47.946,-149.3199,24.3499,0.0000
C01225=-57.387,47.412,47.522,-151.0217,27.5582,0.0000
C01226=-54.990,50.108,47.503,-151.3284,28.0902,0.0000
C01227=-52.606,52.606,47.516,-149.9647,26.5896,0.0000
C01228=-50.108,54.990,47.503,-148.6870,25.0415,0.0000
C01229=-47.412,57.387,47.522,-149.1829,25.4372,0.0000
C01230=-44.975,60.171,47.946,-152.2461,27.7011,0.0000
C01231=-44.675,62.766,49.019,-154.7869,28.9480,0.0000
C01232=-45.859,65.749,50.519,-157.1002,29.7260,0.0000
C01233=-47.903,69.367,52.090,-160.1822,30.3186,0.0000
C01234=-50.285,73.401,53.317,-165.1529,30.3518,0.0000
C01235=-52.213,77.409,53.931,-173.7151,27.6520,0.0000
C01236=-52.061,81.773,54.258,177.7005,15.3195,0.0000
C01237=-49.741,85.881,54.525,177.7942,7.3164,0.0000
C01238=-45.636,88.910,54.796,178.3978,4.5245,0.0000
C01239=-40.787,91.296,54.976,178.6769,3.5372,0.0000
C01240=-35.715,93.397,54.976,-178.4311,-3.4353,0.0000
C01241=-30.600,95.138,54.796,-177.9269,-4.3294,0.0000
C01242=-25.555,95.900,54.525,-176.3598,-6.7215,0.0000
C01243=-21.009,94.635,54.258,-170.6048,-12.3676,0.0000
C01244=-17.816,91.657,53.931,-155.7436,-15.0464,0.0000
C01245=-16.346,87.459,53.317,-148.3749,-11.5926,0.0000
C01246=-15.177,82.922,52.090,-145.2254,-8.6275,0.0000
C01247=-14.064,78.919,50.519,-143.6103,-6.4121,0.0000
C01248=-12.792,75.972,49.019,-142.5753,-4.5119,0.0000
C01249=-10.745,74.349,47.946,-141.6346,-2.1298,0.0000
C01250=-7.053,74.105,47.522,-140.8743,1.3417,0.0000
C01251=-3.453,74.315,47.503,-140.7572,1.9283,0.0000
C01252=0.000,74.396,47.516,-140.7285,-0.0001,0.0000
C01253=0.000,73.003,49.219,-140.7893,-0.0001,0.0000
C01254=3.325,72.927,49.205,-140.8175,-1.9051,0.0000
C01255=6.839,72.729,49.225,-140.9341,-1.2745,0.0000
C01256=10.483,73.017,49.677,-141.7015,2.2500,0.0000
C01257=12.469,74.753,50.822,-142.6316,4.6198,0.0000
C01258=13.691,77.880,52.422,-143.6589,6.5325,0.0000
C01259=14.768,82.123,54.099,-145.3237,8.8372,0.0000
C01260=15.905,86.934,55.407,-148.7673,12.0143,0.0000
C01261=17.335,91.395,56.062,-157.5762,15.5221,0.0000
C01262=20.556,94.581,56.410,-173.1817,10.4947,0.0000
C01263=25.196,95.965,56.695,-177.7245,4.7775,0.0000
C01264=30.373,95.213,56.983,-178.8087,2.7642,0.0000
C01265=35.638,93.426,57.174,-179.1081,2.1395,0.0000
C01266=40.862,91.262,57.174,179.1171,-2.1432,0.0000
C01267=45.849,88.802,56.983,178.8861,-2.7962,0.0000
C01268=50.042,85.674,56.695,178.2217,-4.9836,0.0000
C01269=52.343,81.414,56.410,177.2877,-12.2009,0.0000
C01270=52.368,76.884,56.062,-175.4639,-26.6872,0.0000
C01271=50.225,72.718,55.407,-165.8129,-30.3847,0.0000
C01272=47.627,68.512,54.099,-160.4292,-30.4081,0.0000
C01273=45.389,64.750,52.422,-157.2332,-29.7852,0.0000
C01274=44.041,61.675,50.822,-154.9152,-28.9947,0.0000
C01275=44.219,59.044,49.677,-152.3901,-27.7528,0.0000
C01276=46.591,56.263,49.225,-149.2806,-25.4543,0.0000
C01277=49.216,53.919,49.205,-148.7554,-25.0235,0.0000
C01278=51.621,51.621,49.219,-150.0183,-26.5522,0.0000
C01279=53.919,49.216,49.205,-151.3655,-28.0347,0.0000
C01280=56.263,46.591,49.225,-151.0265,-27.4666,0.0000
C01281=59.044,44.219,49.677,-149.2976,-24.2130,0.0000
C01282=61.675,44.041,50.822,-148.5375,-21.7663,0.0000
C01283=64.750,45.389,52.422,-148.1711,-19.6249,0.0000
C01284=68.512,47.627,54.099,-148.0825,-16.7920,0.0000
C01285=72.718,50.225,55.407,-148.8352,-12.2065,0.0000
C01286=76.884,52.368,56.062,-153.2403,-4.0524,0.0000
C01287=81.414,52.343,56.410,-167.7858,2.6510,0.0000
C01288=85.674,50.042,56.695,-175.0140,1.7716,0.0000
C01289=88.802,45.849,56.983,-177.2032,1.1126,0.0000
C01290=91.262,40.862,57.174,-177.8566,0.8823,0.0000
C01291=93.426,35.638,57.174,177.8603,-0.8913,0.0000
C01292=95.213,30.373,56.983,177.2352,-1.1899,0.0000
C01293=95.965,25.196,56.695,175.2187,-2.2675,0.0000
C01294=94.581,20.556,56.410,169.4322,-6.7038,0.0000
C01295=91.395,17.335,56.062,163.2767,-21.5641,0.0000
C01296=86.934,15.905,55.407,166.0236,-30.4747,0.0000
C01297=82.123,14.768,54.099,169.2944,-34.2070,0.0000
C01298=77.880,13.691,52.422,171.9090,-36.0679,0.0000
C01299=74.753,12.469,50.822,174.1944,-37.2264,0.0000
C01300=73.017,10.483,49.677,177.1339,-38.2636,0.0000
C01301=72.729,6.839,49.225,-178.3587,-39.0544,0.0000
C01302=72.927,3.325,49.205,-177.5428,-39.1567,0.0000
C01303=73.003,0.000,49.219,-179.9998,-39.2107,0.0000
C01304=72.927,-3.325,49.205,177.5428,-39.1567,0.0000
C01305=72.729,-6.839,49.225,178.3601,-39.0543,0.0000
C01306=73.017,-10.483,49.677,-177.1334,-38.2635,0.0000
C01307=74.753,-12.469,50.822,-174.1943,-37.2263,0.0000
C01308=77.880,-13.691,52.422,-171.9092,-36.0680,0.0000
C01309=82.123,-14.768,54.099,-169.2947,-34.2072,0.0000
C01310=86.934,-15.905,55.407,-166.0241,-30.4751,0.0000
C01311=91.395,-17.335,56.062,-163.2768,-21.5645,0.0000
C01312=94.581,-20.556,56.410,-169.4322,-6.7038,0.0000
C01313=95.965,-25.196,56.695,-175.2187,-2.2675,0.0000
C01314=95.213,-30.373,56.983,-177.2352,-1.1899,0.0000
C01315=93.426,-35.638,57.174,-177.8603,-0.8913,0.0000
C01316=91.262,-40.862,57.174,177.8566,0.8823,0.0000
C01317=88.802,-45.849,56.983,177.2032,1.1126,0.0000
C01318=85.674,-50.042,56.695,175.0140,1.7716,0.0000
C01319=81.414,-52.343,56.410,167.7858,2.6510,0.0000
C01320=76.884,-52.368,56.062,153.2406,-4.0520,0.0000
C01321=72.718,-50.225,55.407,148.8352,-12.2059,0.0000
C01322=68.512,-47.627,54.099,148.0824,-16.7917,0.0000
C01323=64.750,-45.389,52.422,148.1710,-19.6248,0.0000
C01324=61.675,-44.041,50.822,148.5375,-21.7664,0.0000
C01325=59.044,-44.219,49.677,149.2978,-24.2134,0.0000
C01326=56.263,-46.591,49.225,151.0271,-27.4675,0.0000
C01327=53.919,-49.216,49.205,151.3655,-28.0346,0.0000
C01328=51.621,-51.621,49.219,150.0185,-26.5524,0.0000
C01329=49.216,-53.919,49.205,148.7554,-25.0235,0.0000
C01330=46.591,-56.263,49.225,149.2815,-25.4551,0.0000
C01331=44.219,-59.044,49.677,152.3905,-27.7531,0.0000
C01332=44.041,-61.675,50.822,154.9153,-28.9947,0.0000
C01333=45.389,-64.750,52.422,157.2330,-29.7852,0.0000
C01334=47.627,-68.512,54.099,160.4288,-30.4080,0.0000
C01335=50.225,-72.718,55.407,165.8123,-30.3846,0.0000
C01336=52.368,-76.884,56.062,175.4635,-26.6874,0.0000
C01337=52.343,-81.414,56.410,-177.2877,-12.2009,0.0000
C01338=50.042,-85.674,56.695,-178.2217,-4.9836,0.0000
C01339=45.849,-88.802,56.983,-178.8861,-2.7962,0.0000
C01340=40.862,-91.262,57.174,-179.1171,-2.1432,0.0000
C01341=35.638,-93.426,57.174,179.1081,2.1395,0.0000
C01342=30.373,-95.213,56.983,178.8087,2.7642,0.0000
C01343=25.196,-95.965,56.695,177.7245,4.7775,0.0000
C01344=20.556,-94.581,56.410,173.1817,10.4947,0.0000
C01345=17.335,-91.395,56.062,157.5762,15.5221,0.0000
C01346=15.905,-86.934,55.407,148.7673,12.0143,0.0000
C01347=14.768,-82.123,54.099,145.3237,8.8372,0.0000
C01348=13.691,-77.880,52.422,143.6589,6.5325,0.0000
C01349=12.469,-74.753,50.822,142.6316,4.6198,0.0000
C01350=10.483,-73.017,49.677,141.7015,2.2500,0.0000
C01351=6.839,-72.729,49.225,140.9341,-1.2745,0.0000
C01352=3.325,-72.927,49.205,140.8175,-1.9051,0.0000
C01353=0.000,-73.003,49.219,140.7893,-0.0001,0.0000
C01354=0.000,-73.003,49.219,140.7893,-0.0001,0.0000
C01355=-3.325,-72.927,49.205,140.8175,1.9052,0.0000
C01356=-6.839,-72.729,49.225,140.9342,1.2734,0.0000
C01357=-10.483,-73.017,49.677,141.7017,-2.2504,0.0000
C01358=-12.469,-74.753,50.822,142.6316,-4.6199,0.0000
C01359=-13.691,-77.880,52.422,143.6589,-6.5324,0.0000
C01360=-14.768,-82.123,54.099,145.3236,-8.8369,0.0000
C01361=-15.905,-86.934,55.407,148.7669,-12.0139,0.0000
C01362=-17.335,-91.395,56.062,157.5758,-15.5220,0.0000
C01363=-20.556,-94.581,56.410,173.1817,-10.4947,0.0000
C01364=-25.196,-95.965,56.695,177.7245,-4.7775,0.0000
C01365=-30.373,-95.213,56.983,178.8087,-2.7642,0.0000
C01366=-35.638,-93.426,57.174,179.1081,-2.1395,0.0000
C01367=-40.862,-91.262,57.174,-179.1171,2.1432,0.0000
C01368=-45.849,-88.802,56.983,-178.8861,2.7962,0.0000
C01369=-50.042,-85.674,56.695,-178.2217,4.9836,0.0000
C01370=-52.343,-81.414,56.410,-177.2877,12.2009,0.0000
C01371=-52.368,-76.884,56.062,175.4639,26.6872,0.0000
C01372=-50.225,-72.718,55.407,165.8129,30.3847,0.0000
C01373=-47.627,-68.512,54.099,160.4292,30.4081,0.0000
C01374=-45.389,-64.750,52.422,157.2332,29.7852,0.0000
C01375=-44.041,-61.675,50.822,154.9152,28.9947,0.0000
C01376=-44.219,-59.044,49.677,152.3901,27.7528,0.0000
C01377=-46.591,-56.263,49.225,149.2806,25.4543,0.0000
C01378=-49.216,-53.919,49.205,148.7554,25.0235,0.0000
C01379=-51.621,-51.621,49.219,150.0183,26.5522,0.0000
C01380=-53.919,-49.216,49.205,151.3655,28.0347,0.0000
C01381=-56.263,-46.591,49.225,151.0265,27.4666,0.0000
C01382=-59.044,-44.219,49.677,149.2976,24.2130,0.0000
C01383=-61.675,-44.041,50.822,148.5375,21.7663,0.0000
C01384=-64.750,-45.389,52.422,148.1711,19.6249,0.0000
C01385=-68.512,-47.627,54.099,148.0825,16.7920,0.0000
C01386=-72.718,-50.225,55.407,148.8352,12.2065,0.0000
C01387=-76.884,-52.368,56.062,153.2403,4.0524,0.0000
C01388=-81.414,-52.343,56.410,167.7858,-2.6510,0.0000
C01389=-85.674,-50.042,56.695,175.0140,-1.7716,0.0000
C01390=-88.802,-45.849,56.983,177.2032,-1.1126,0.0000
C01391=-91.262,-40.862,57.174,177.8566,-0.8823,0.0000
C01392=-93.426,-35.638,57.174,-177.8603,0.8913,0.0000
C01393=-95.213,-30.373,56.983,-177.2352,1.1899,0.0000
C01394=-95.965,-25.196,56.695,-175.2187,2.2675,0.0000
C01395=-94.581,-20.556,56.410,-169.4322,6.7038,0.0000
C01396=-91.395,-17.335,56.062,-163.2767,21.5641,0.0000
C01397=-86.934,-15.905,55.407,-166.0236,30.4747,0.0000
C01398=-82.123,-14.768,54.099,-169.2944,34.2070,0.0000
C01399=-77.880,-13.691,52.422,-171.9090,36.0679,0.0000
C01400=-74.753,-12.469,50.822,-174.1944,37.2264,0.0000
C01401=-73.017,-10.483,49.677,-177.1339,38.2636,0.0000
C01402=-72.729,-6.839,49.225,178.3587,39.0544,0.0000
C01403=-72.927,-3.325,49.205,177.5428,39.1567,0.0000
C01404=-73.003,0.000,49.219,179.9998,39.2107,0.0000
C01405=-72.927,3.325,49.205,-177.5428,39.1567,0.0000
C01406=-72.729,6.839,49.225,-178.3601,39.0543,0.0000
C01407=-73.017,10.483,49.677,177.1334,38.2635,0.0000
C01408=-74.753,12.469,50.822,174.1943,37.2263,0.0000
C01409=-77.880,13.691,52.422,171.9092,36.0680,0.0000
C01410=-82.123,14.768,54.099,169.2947,34.2072,0.0000
C01411=-86.934,15.905,55.407,166.0241,30.4751,0.0000
C01412=-91.395,17.335,56.062,163.2768,21.5645,0.0000
C01413=-94.581,20.556,56.410,169.4322,6.7038,0.0000
C01414=-95.965,25.196,56.695,175.2187,2.2675,0.0000
C01415=-95.213,30.373,56.983,177.2352,1.1899,0.0000
C01416=-93.426,35.638,57.174,177.8603,0.8913,0.0000
C01417=-91.262,40.862,57.174,-177.8566,-0.8823,0.0000
C01418=-88.802,45.849,56.983,-177.2032,-1.1126,0.0000
C01419=-85.674,50.042,56.695,-175.0140,-1.7716,0.0000
C01420=-81.414,52.343,56.410,-167.7858,-2.6510,0.0000
C01421=-76.884,52.368,56.062,-153.2406,4.0520,0.0000
C01422=-72.718,50.225,55.407,-148.8352,12.2059,0.0000
C01423=-68.512,47.627,54.099,-148.0824,16.7917,0.0000
C01424=-64.750,45.389,52.422,-148.1710,19.6248,0.0000
C01425=-61.675,44.041,50.822,-148.5375,21.7664,0.0000
C01426=-59.044,44.219,49.677,-149.2978,24.2134,0.0000
C01427=-56.263,46.591,49.225,-151.0271,27.4675,0.0000
C01428=-53.919,49.216,49.205,-151.3655,28.0346,0.0000
C01429=-51.621,51.621,49.219,-150.0185,26.5524,0.0000
C01430=-49.216,53.919,49.205,-148.7554,25.0235,0.0000
C01431=-46.591,56.263,49.225,-149.2815,25.4551,0.0000
C01432=-44.219,59.044,49.677,-152.3905,27.7531,0.0000
C01433=-44.041,61.675,50.822,-154.9153,28.9947,0.0000
C01434=-45.389,64.750,52.422,-157.2330,29.7852,0.0000
C01435=-47.627,68.512,54.099,-160.4288,30.4080,0.0000
C01436=-50.225,72.718,55.407,-165.8123,30.3846,0.0000
C01437=-52.368,76.884,56.062,-175.4635,26.6874,0.0000
C01438=-52.343,81.414,56.410,177.2877,12.2009,0.0000
C01439=-50.042,85.674,56.695,178.2217,4.9836,0.0000
C01440=-45.849,88.802,56.983,178.8861,2.7962,0.0000
C01441=-40.862,91.262,57.174,179.1171,2.1432,0.0000
C01442=-35.638,93.426,57.174,-179.1081,-2.1395,0.0000
C01443=-30.373,95.213,56.983,-178.8087,-2.7642,0.0000
C01444=-25.196,95.965,56.695,-177.7245,-4.7775,0.0000
C01445=-20.556,94.581,56.410,-173.1817,-10.4947,0.0000
C01446=-17.335,91.395,56.062,-157.5758,-15.5220,0.0000
C01447=-15.905,86.934,55.407,-148.7669,-12.0139,0.0000
C01448=-14.768,82.123,54.099,-145.3236,-8.8369,0.0000
C01449=-13.691,77.880,52.422,-143.6589,-6.5324,0.0000
C01450=-12.469,74.753,50.822,-142.6316,-4.6199,0.0000
C01451=-10.483,73.017,49.677,-141.7017,-2.2504,0.0000
C01452=-6.839,72.729,49.225,-140.9342,1.2734,0.0000
C01453=-3.325,72.927,49.205,-140.8175,1.9052,0.0000
C01454=0.000,73.003,49.219,-140.7893,-0.0001,0.0000
C01455=0.000,71.612,50.923,-140.8954,-0.0002,0.0000
C01456=3.198,71.541,50.909,-140.9230,-1.8787,0.0000
C01457=6.625,71.354,50.929,-141.0390,-1.2107,0.0000
C01458=10.220,71.688,51.410,-141.8121,2.3568,0.0000
C01459=12.146,73.537,52.627,-142.7298,4.7102,0.0000
C01460=13.319,76.847,54.328,-143.7495,6.6367,0.0000
C01461=14.363,81.331,56.111,-145.4725,9.0405,0.0000
C01462=15.469,86.415,57.500,-149.2812,12.4578,0.0000
C01463=16.861,91.137,58.195,-160.1229,15.8031,0.0000
C01464=20.110,94.527,58.564,-175.5000,8.1577,0.0000
C01465=24.842,96.029,58.865,-178.8015,2.8497,0.0000
C01466=30.149,95.287,59.171,-179.5109,1.2561,0.0000
C01467=35.562,93.456,59.373,-179.6626,0.8844,0.0000
C01468=40.937,91.230,59.373,179.6132,-0.8639,0.0000
C01469=46.059,88.697,59.171,179.4575,-1.2340,0.0000
C01470=50.337,85.469,58.865,178.8306,-2.8617,0.0000
C01471=52.621,81.060,58.564,177.3647,-8.9316,0.0000
C01472=52.521,76.366,58.195,-177.5470,-25.0811,0.0000
C01473=50.167,72.043,57.500,-166.5883,-30.3473,0.0000
C01474=47.354,67.666,56.111,-160.7140,-30.4589,0.0000
C01475=44.921,63.757,54.328,-157.3902,-29.8046,0.0000
C01476=43.410,60.587,52.627,-155.0673,-29.0009,0.0000
C01477=43.464,57.918,51.410,-152.5630,-27.7666,0.0000
C01478=45.770,55.140,50.929,-149.4158,-25.4411,0.0000
C01479=48.325,52.849,50.909,-148.8657,-24.9808,0.0000
C01480=50.637,50.637,50.923,-150.1120,-26.4871,0.0000
C01481=52.848,48.326,50.909,-151.4405,-27.9485,0.0000
C01482=55.140,45.770,50.930,-151.0748,-27.3516,0.0000
C01483=57.918,43.464,51.410,-149.3224,-24.0610,0.0000
C01484=60.587,43.410,52.627,-148.5625,-21.6351,0.0000
C01485=63.757,44.921,54.328,-148.1804,-19.4875,0.0000
C01486=67.666,47.354,56.111,-148.0754,-16.5414,0.0000
C01487=72.043,50.167,57.500,-148.9572,-11.5472,0.0000
C01488=76.366,52.521,58.195,-154.8985,-2.2219,0.0000
C01489=81.060,52.621,58.564,-171.0591,2.6033,0.0000
C01490=85.469,50.337,58.865,-177.1377,1.1679,0.0000
C01491=88.697,46.059,59.171,-178.7659,0.5424,0.0000
C01492=91.230,40.937,59.373,-179.1361,0.3868,0.0000
C01493=93.456,35.562,59.373,179.1156,-0.3374,0.0000
C01494=95.287,30.149,59.171,178.7438,-0.4890,0.0000
C01495=96.029,24.842,58.865,177.1497,-1.1970,0.0000
C01496=94.527,20.110,58.564,171.8174,-4.4543,0.0000
C01497=91.137,16.861,58.195,163.2503,-19.0961,0.0000
C01498=86.415,15.469,57.500,165.5879,-29.9205,0.0000
C01499=81.331,14.363,56.111,169.0692,-34.0393,0.0000
C01500=76.847,13.319,54.328,171.7901,-35.9695,0.0000
C01501=73.537,12.146,52.627,174.0888,-37.1231,0.0000
C01502=71.688,10.220,51.410,177.0026,-38.1498,0.0000
C01503=71.354,6.625,50.929,-178.4432,-38.9507,0.0000
C01504=71.541,3.198,50.909,-177.5805,-39.0520,0.0000
C01505=71.612,0.000,50.923,-179.9997,-39.1046,0.0000
C01506=71.541,-3.198,50.909,177.5804,-39.0520,0.0000
C01507=71.354,-6.626,50.930,178.4446,-38.9506,0.0000
C01508=71.688,-10.221,51.410,-177.0020,-38.1497,0.0000
C01509=73.537,-12.146,52.627,-174.0887,-37.1230,0.0000
C01510=76.847,-13.319,54.328,-171.7902,-35.9695,0.0000
C01511=81.331,-14.363,56.111,-169.0696,-34.0395,0.0000
C01512=86.415,-15.469,57.500,-165.5884,-29.9209,0.0000
C01513=91.137,-16.861,58.195,-163.2503,-19.0965,0.0000
C01514=94.527,-20.110,58.564,-171.8174,-4.4543,0.0000
C01515=96.029,-24.842,58.865,-177.1497,-1.1970,0.0000
C01516=95.287,-30.149,59.171,-178.7438,-0.4890,0.0000
C01517=93.456,-35.562,59.373,-179.1156,-0.3374,0.0000
C01518=91.230,-40.937,59.373,179.1361,0.3868,0.0000
C01519=88.697,-46.059,59.171,178.7659,0.5424,0.0000
C01520=85.469,-50.337,58.865,177.1377,1.1679,0.0000
C01521=81.060,-52.621,58.564,171.0591,2.6033,0.0000
C01522=76.366,-52.521,58.195,154.8987,-2.2216,0.0000
C01523=72.043,-50.167,57.500,148.9573,-11.5466,0.0000
C01524=67.666,-47.354,56.111,148.0753,-16.5410,0.0000
C01525=63.757,-44.921,54.328,148.1803,-19.4874,0.0000
C01526=60.587,-43.410,52.627,148.5625,-21.6352,0.0000
C01527=57.918,-43.464,51.410,149.3226,-24.0615,0.0000
C01528=55.140,-45.770,50.929,151.0754,-27.3525,0.0000
C01529=52.849,-48.325,50.909,151.4405,-27.9484,0.0000
C01530=50.637,-50.637,50.923,150.1122,-26.4875,0.0000
C01531=48.326,-52.848,50.909,148.8655,-24.9807,0.0000
C01532=45.770,-55.140,50.930,149.4167,-25.4419,0.0000
C01533=43.464,-57.918,51.410,152.5634,-27.7669,0.0000
C01534=43.410,-60.587,52.627,155.0675,-29.0010,0.0000
C01535=44.921,-63.757,54.328,157.3901,-29.8046,0.0000
C01536=47.354,-67.666,56.111,160.7137,-30.4588,0.0000
C01537=50.167,-72.043,57.500,166.5876,-30.3473,0.0000
C01538=52.521,-76.366,58.195,177.5467,-25.0813,0.0000
C01539=52.621,-81.060,58.564,-177.3647,-8.9316,0.0000
C01540=50.337,-85.469,58.865,-178.8306,-2.8617,0.0000
C01541=46.059,-88.697,59.171,-179.4575,-1.2340,0.0000
C01542=40.937,-91.230,59.373,-179.6132,-0.8639,0.0000
C01543=35.562,-93.456,59.373,179.6626,0.8844,0.0000
C01544=30.149,-95.287,59.171,179.5109,1.2561,0.0000
C01545=24.842,-96.029,58.865,178.8015,2.8497,0.0000
C01546=20.110,-94.527,58.564,175.5000,8.1577,0.0000
C01547=16.861,-91.137,58.195,160.1229,15.8031,0.0000
C01548=15.469,-86.415,57.500,149.2812,12.4578,0.0000
C01549=14.363,-81.331,56.111,145.4725,9.0405,0.0000
C01550=13.319,-76.847,54.328,143.7495,6.6367,0.0000
C01551=12.146,-73.537,52.627,142.7298,4.7102,0.0000
C01552=10.220,-71.688,51.410,141.8121,2.3568,0.0000
C01553=6.625,-71.354,50.929,141.0390,-1.2107,0.0000
C01554=3.198,-71.541,50.909,140.9230,-1.8787,0.0000
C01555=0.000,-71.612,50.923,140.8954,-0.0002,0.0000
C01556=0.000,-71.612,50.923,140.8954,-0.0002,0.0000
C01557=-3.198,-71.541,50.909,140.9230,1.8788,0.0000
C01558=-6.626,-71.354,50.930,141.0391,1.2096,0.0000
C01559=-10.221,-71.688,51.410,141.8122,-2.3572,0.0000
C01560=-12.146,-73.537,52.627,142.7299,-4.7103,0.0000
C01561=-13.319,-76.847,54.328,143.7495,-6.6366,0.0000
C01562=-14.363,-81.331,56.111,145.4723,-9.0401,0.0000
C01563=-15.469,-86.415,57.500,149.2808,-12.4574,0.0000
C01564=-16.861,-91.137,58.195,160.1225,-15.8031,0.0000
C01565=-20.110,-94.527,58.564,175.5000,-8.1577,0.0000
C01566=-24.842,-96.029,58.865,178.8015,-2.8497,0.0000
C01567=-30.149,-95.287,59.171,179.5109,-1.2561,0.0000
C01568=-35.562,-93.456,59.373,179.6626,-0.8844,0.0000
C01569=-40.937,-91.230,59.373,-179.6132,0.8639,0.0000
C01570=-46.059,-88.697,59.171,-179.4575,1.2340,0.0000
C01571=-50.337,-85.469,58.865,-178.8306,2.8617,0.0000
C01572=-52.621,-81.060,58.564,-177.3647,8.9316,0.0000
C01573=-52.521,-76.366,58.195,177.5470,25.0811,0.0000
C01574=-50.167,-72.043,57.500,166.5883,30.3473,0.0000
C01575=-47.354,-67.666,56.111,160.7140,30.4589,0.0000
C01576=-44.921,-63.757,54.328,157.3902,29.8046,0.0000
C01577=-43.410,-60.587,52.627,155.0673,29.0009,0.0000
C01578=-43.464,-57.918,51.410,152.5630,27.7666,0.0000
C01579=-45.770,-55.140,50.929,149.4158,25.4411,0.0000
C01580=-48.325,-52.849,50.909,148.8657,24.9808,0.0000
C01581=-50.637,-50.637,50.923,150.1120,26.4871,0.0000
C01582=-52.848,-48.326,50.909,151.4405,27.9485,0.0000
C01583=-55.140,-45.770,50.930,151.0748,27.3516,0.0000
C01584=-57.918,-43.464,51.410,149.3224,24.0610,0.0000
C01585=-60.587,-43.410,52.627,148.5625,21.6351,0.0000
C01586=-63.757,-44.921,54.328,148.1804,19.4875,0.0000
C01587=-67.666,-47.354,56.111,148.0754,16.5414,0.0000
C01588=-72.043,-50.167,57.500,148.9572,11.5472,0.0000
C01589=-76.366,-52.521,58.195,154.8985,2.2219,0.0000
C01590=-81.060,-52.621,58.564,171.0591,-2.6033,0.0000
C01591=-85.469,-50.337,58.865,177.1377,-1.1679,0.0000
C01592=-88.697,-46.059,59.171,178.7659,-0.5424,0.0000
C01593=-91.230,-40.937,59.373,179.1361,-0.3868,0.0000
C01594=-93.456,-35.562,59.373,-179.1156,0.3374,0.0000
C01595=-95.287,-30.149,59.171,-178.7438,0.4890,0.0000
C01596=-96.029,-24.842,58.865,-177.1497,1.1970,0.0000
C01597=-94.527,-20.110,58.564,-171.8174,4.4543,0.0000
C01598=-91.137,-16.861,58.195,-163.2503,19.0961,0.0000
C01599=-86.415,-15.469,57.500,-165.5879,29.9205,0.0000
C01600=-81.331,-14.363,56.111,-169.0692,34.0393,0.0000
C01601=-76.847,-13.319,54.328,-171.7901,35.9695,0.0000
C01602=-73.537,-12.146,52.627,-174.0888,37.1231,0.0000
C01603=-71.688,-10.220,51.410,-177.0026,38.1498,0.0000
C01604=-71.354,-6.625,50.929,178.4432,38.9507,0.0000
C01605=-71.541,-3.198,50.909,177.5805,39.0520,0.0000
C01606=-71.612,0.000,50.923,179.9997,39.1046,0.0000
C01607=-71.541,3.198,50.909,-177.5804,39.0520,0.0000
C01608=-71.354,6.626,50.930,-178.4446,38.9506,0.0000
C01609=-71.688,10.221,51.410,177.0020,38.1497,0.0000
C01610=-73.537,12.146,52.627,174.0887,37.1230,0.0000
C01611=-76.847,13.319,54.328,171.7902,35.9695,0.0000
C01612=-81.331,14.363,56.111,169.0696,34.0395,0.0000
C01613=-86.415,15.469,57.500,165.5884,29.9209,0.0000
C01614=-91.137,16.861,58.195,163.2503,19.0965,0.0000
C01615=-94.527,20.110,58.564,171.8174,4.4543,0.0000
C01616=-96.029,24.842,58.865,177.1497,1.1970,0.0000
C01617=-95.287,30.149,59.171,178.7438,0.4890,0.0000
C01618=-93.456,35.562,59.373,179.1156,0.3374,0.0000
C01619=-91.230,40.937,59.373,-179.1361,-0.3868,0.0000
C01620=-88.697,46.059,59.171,-178.7659,-0.5424,0.0000
C01621=-85.469,50.337,58.865,-177.1377,-1.1679,0.0000
C01622=-81.060,52.621,58.564,-171.0591,-2.6033,0.0000
C01623=-76.366,52.521,58.195,-154.8987,2.2216,0.0000
C01624=-72.043,50.167,57.500,-148.9573,11.5466,0.0000
C01625=-67.666,47.354,56.111,-148.0753,16.5410,0.0000
C01626=-63.757,44.921,54.328,-148.1803,19.4874,0.0000
C01627=-60.587,43.410,52.627,-148.5625,21.6352,0.0000
C01628=-57.918,43.464,51.410,-149.3226,24.0615,0.0000
C01629=-55.140,45.770,50.929,-151.0754,27.3525,0.0000
C01630=-52.849,48.325,50.909,-151.4405,27.9484,0.0000
C01631=-50.637,50.637,50.923,-150.1122,26.4875,0.0000
C01632=-48.326,52.848,50.909,-148.8655,24.9807,0.0000
C01633=-45.770,55.140,50.930,-149.4167,25.4419,0.0000
C01634=-43.464,57.918,51.410,-152.5634,27.7669,0.0000
C01635=-43.410,60.587,52.627,-155.0675,29.0010,0.0000
C01636=-44.921,63.757,54.328,-157.3901,29.8046,0.0000
C01637=-47.354,67.666,56.111,-160.7137,30.4588,0.0000
C01638=-50.167,72.043,57.500,-166.5876,30.3473,0.0000
C01639=-52.521,76.366,58.195,-177.5467,25.0813,0.0000
C01640=-52.621,81.060,58.564,177.3647,8.9316,0.0000
C01641=-50.337,85.469,58.865,178.8306,2.8617,0.0000
C01642=-46.059,88.697,59.171,179.4575,1.2340,0.0000
C01643=-40.937,91.230,59.373,179.6132,0.8639,0.0000
C01644=-35.562,93.456,59.373,-179.6626,-0.8844,0.0000
C01645=-30.149,95.287,59.171,-179.5109,-1.2561,0.0000
C01646=-24.842,96.029,58.865,-178.8015,-2.8497,0.0000
C01647=-20.110,94.527,58.564,-175.5000,-8.1577,0.0000
C01648=-16.861,91.137,58.195,-160.1225,-15.8031,0.0000
C01649=-15.469,86.415,57.500,-149.2808,-12.4574,0.0000
C01650=-14.363,81.331,56.111,-145.4723,-9.0401,0.0000
C01651=-13.319,76.847,54.328,-143.7495,-6.6366,0.0000
C01652=-12.146,73.537,52.627,-142.7299,-4.7103,0.0000
C01653=-10.221,71.688,51.410,-141.8122,-2.3572,0.0000
C01654=-6.626,71.354,50.930,-141.0391,1.2096,0.0000
C01655=-3.198,71.541,50.909,-140.9230,1.8788,0.0000
C01656=0.000,71.612,50.923,-140.8954,-0.0002,0.0000
C01657=0.000,70.224,52.630,-141.0463,-0.0003,0.0000
C01658=3.072,70.158,52.615,-141.0733,-1.8491,0.0000
C01659=6.412,69.984,52.637,-141.1884,-1.1514,0.0000
C01660=9.959,70.362,53.146,-141.9656,2.4499,0.0000
C01661=11.825,72.328,54.436,-142.8698,4.7838,0.0000
C01662=12.951,75.822,56.240,-143.8825,6.7262,0.0000
C01663=13.963,80.549,58.128,-145.6744,9.2407,0.0000
C01664=15.041,85.905,59.597,-149.9457,12.9304,0.0000
C01665=16.396,90.884,60.330,-163.7506,15.5606,0.0000
C01666=19.672,94.474,60.719,-177.3628,5.6237,0.0000
C01667=24.496,96.092,61.037,-179.6023,1.0626,0.0000
C01668=29.931,95.359,61.359,179.9514,-0.1374,0.0000
C01669=35.488,93.484,61.571,179.8966,-0.2951,0.0000
C01670=41.009,91.197,61.571,-179.8644,0.2818,0.0000
C01671=46.265,88.593,61.359,-179.9372,0.1316,0.0000
C01672=50.626,85.269,61.037,179.5298,-1.0326,0.0000
C01673=52.893,80.714,60.719,177.8734,-5.8354,0.0000
C01674=52.671,75.858,60.330,-179.9428,-22.3521,0.0000
C01675=50.109,71.379,59.597,-167.5063,-30.2239,0.0000
C01676=47.084,66.830,58.128,-161.0416,-30.4714,0.0000
C01677=44.457,62.772,56.240,-157.5727,-29.7852,0.0000
C01678=42.782,59.505,54.436,-155.2435,-28.9674,0.0000
C01679=42.712,56.796,53.146,-152.7639,-27.7426,0.0000
C01680=44.952,54.020,52.637,-149.5870,-25.3970,0.0000
C01681=47.437,51.781,52.615,-149.0172,-24.9133,0.0000
C01682=49.656,49.656,52.630,-150.2450,-26.3945,0.0000
C01683=51.781,47.437,52.615,-151.5528,-27.8320,0.0000
C01684=54.020,44.952,52.637,-151.1655,-27.2125,0.0000
C01685=56.796,42.711,53.146,-149.3936,-23.8938,0.0000
C01686=59.505,42.782,54.436,-148.6339,-21.4920,0.0000
C01687=62.772,44.457,56.240,-148.2344,-19.3363,0.0000
C01688=66.830,47.084,58.128,-148.1135,-16.2611,0.0000
C01689=71.379,50.109,59.597,-149.1752,-10.7740,0.0000
C01690=75.858,52.671,60.330,-157.6477,-0.0531,0.0000
C01691=80.714,52.893,60.719,-174.1606,2.1156,0.0000
C01692=85.269,50.626,61.037,-178.9674,0.4701,0.0000
C01693=88.593,46.265,61.359,179.8684,-0.0628,0.0000
C01694=91.197,41.009,61.571,179.7182,-0.1356,0.0000
C01695=93.484,35.488,61.571,-179.7049,0.1034,0.0000
C01696=95.359,29.931,61.359,-179.8626,0.0486,0.0000
C01697=96.092,24.496,61.037,178.9374,-0.3977,0.0000
C01698=94.474,19.672,60.719,174.3703,-2.6245,0.0000
C01699=90.884,16.396,60.330,163.8251,-15.6383,0.0000
C01700=85.905,15.041,59.597,165.1443,-29.2171,0.0000
C01701=80.549,13.963,58.128,168.8553,-33.8194,0.0000
C01702=75.822,12.951,56.240,171.6938,-35.8302,0.0000
C01703=72.328,11.825,54.436,174.0078,-36.9792,0.0000
C01704=70.362,9.959,53.146,176.8908,-37.9934,0.0000
C01705=69.984,6.412,52.637,-178.5225,-38.8023,0.0000
C01706=70.158,3.072,52.615,-177.6237,-38.9026,0.0000
C01707=70.224,0.000,52.630,-179.9996,-38.9537,0.0000
C01708=70.158,-3.071,52.615,177.6234,-38.9027,0.0000
C01709=69.984,-6.412,52.637,178.5239,-38.8022,0.0000
C01710=70.362,-9.959,53.146,-176.8902,-37.9933,0.0000
C01711=72.328,-11.825,54.436,-174.0076,-36.9792,0.0000
C01712=75.822,-12.951,56.240,-171.6939,-35.8303,0.0000
C01713=80.549,-13.963,58.128,-168.8556,-33.8196,0.0000
C01714=85.905,-15.041,59.597,-165.1447,-29.2176,0.0000
C01715=90.884,-16.396,60.330,-163.8251,-15.6386,0.0000
C01716=94.474,-19.672,60.719,-174.3703,-2.6245,0.0000
C01717=96.092,-24.496,61.037,-178.9374,-0.3977,0.0000
C01718=95.359,-29.931,61.359,179.8626,0.0486,0.0000
C01719=93.484,-35.488,61.571,179.7049,0.1034,0.0000
C01720=91.197,-41.009,61.571,-179.7182,-0.1356,0.0000
C01721=88.593,-46.265,61.359,-179.8684,-0.0628,0.0000
C01722=85.269,-50.626,61.037,178.9674,0.4701,0.0000
C01723=80.714,-52.893,60.719,174.1606,2.1156,0.0000
C01724=75.858,-52.671,60.330,157.6479,-0.0529,0.0000
C01725=71.379,-50.109,59.597,149.1753,-10.7734,0.0000
C01726=66.830,-47.084,58.128,148.1134,-16.2608,0.0000
C01727=62.772,-44.457,56.240,148.2344,-19.3362,0.0000
C01728=59.505,-42.782,54.436,148.6339,-21.4921,0.0000
C01729=56.796,-42.712,53.146,149.3937,-23.8942,0.0000
C01730=54.020,-44.952,52.637,151.1661,-27.2134,0.0000
C01731=51.781,-47.437,52.615,151.5527,-27.8318,0.0000
C01732=49.656,-49.656,52.630,150.2454,-26.3949,0.0000
C01733=47.437,-51.781,52.615,149.0170,-24.9132,0.0000
C01734=44.952,-54.020,52.637,149.5878,-25.3979,0.0000
C01735=42.711,-56.796,53.146,152.7643,-27.7428,0.0000
C01736=42.782,-59.505,54.436,155.2436,-28.9675,0.0000
C01737=44.457,-62.772,56.240,157.5727,-29.7852,0.0000
C01738=47.084,-66.830,58.128,161.0412,-30.4713,0.0000
C01739=50.109,-71.379,59.597,167.5055,-30.2239,0.0000
C01740=52.671,-75.858,60.330,179.9426,-22.3523,0.0000
C01741=52.893,-80.714,60.719,-177.8734,-5.8354,0.0000
C01742=50.626,-85.269,61.037,-179.5298,-1.0326,0.0000
C01743=46.265,-88.593,61.359,179.9372,0.1316,0.0000
C01744=41.009,-91.197,61.571,179.8644,0.2818,0.0000
C01745=35.488,-93.484,61.571,-179.8966,-0.2951,0.0000
C01746=29.931,-95.359,61.359,-179.9514,-0.1374,0.0000
C01747=24.496,-96.092,61.037,179.6023,1.0626,0.0000
C01748=19.672,-94.474,60.719,177.3628,5.6237,0.0000
C01749=16.396,-90.884,60.330,163.7506,15.5606,0.0000
C01750=15.041,-85.905,59.597,149.9457,12.9304,0.0000
C01751=13.963,-80.549,58.128,145.6744,9.2407,0.0000
C01752=12.951,-75.822,56.240,143.8825,6.7262,0.0000
C01753=11.825,-72.328,54.436,142.8698,4.7838,0.0000
C01754=9.959,-70.362,53.146,141.9656,2.4499,0.0000
C01755=6.412,-69.984,52.637,141.1884,-1.1514,0.0000
C01756=3.072,-70.158,52.615,141.0733,-1.8491,0.0000
C01757=0.000,-70.224,52.630,141.0463,-0.0003,0.0000
C01758=0.000,-70.224,52.630,141.0463,-0.0003,0.0000
C01759=-3.071,-70.158,52.615,141.0732,1.8493,0.0000
C01760=-6.412,-69.984,52.637,141.1885,1.1503,0.0000
C01761=-9.959,-70.362,53.146,141.9657,-2.4503,0.0000
C01762=-11.825,-72.328,54.436,142.8698,-4.7839,0.0000
C01763=-12.951,-75.822,56.240,143.8825,-6.7261,0.0000
C01764=-13.963,-80.549,58.128,145.6743,-9.2404,0.0000
C01765=-15.041,-85.905,59.597,149.9453,-12.9300,0.0000
C01766=-16.396,-90.884,60.330,163.7502,-15.5606,0.0000
C01767=-19.672,-94.474,60.719,177.3628,-5.6237,0.0000
C01768=-24.496,-96.092,61.037,179.6023,-1.0626,0.0000
C01769=-29.931,-95.359,61.359,-179.9514,0.1374,0.0000
C01770=-35.488,-93.484,61.571,-179.8966,0.2951,0.0000
C01771=-41.009,-91.197,61.571,179.8644,-0.2818,0.0000
C01772=-46.265,-88.593,61.359,179.9372,-0.1316,0.0000
C01773=-50.626,-85.269,61.037,-179.5298,1.0326,0.0000
C01774=-52.893,-80.714,60.719,-177.8734,5.8354,0.0000
C01775=-52.671,-75.858,60.330,179.9428,22.3521,0.0000
C01776=-50.109,-71.379,59.597,167.5063,30.2239,0.0000
C01777=-47.084,-66.830,58.128,161.0416,30.4714,0.0000
C01778=-44.457,-62.772,56.240,157.5727,29.7852,0.0000
C01779=-42.782,-59.505,54.436,155.2435,28.9674,0.0000
C01780=-42.712,-56.796,53.146,152.7639,27.7426,0.0000
C01781=-44.952,-54.020,52.637,149.5870,25.3970,0.0000
C01782=-47.437,-51.781,52.615,149.0172,24.9133,0.0000
C01783=-49.656,-49.656,52.630,150.2450,26.3945,0.0000
C01784=-51.781,-47.437,52.615,151.5528,27.8320,0.0000
C01785=-54.020,-44.952,52.637,151.1655,27.2125,0.0000
C01786=-56.796,-42.711,53.146,149.3936,23.8938,0.0000
C01787=-59.505,-42.782,54.436,148.6339,21.4920,0.0000
C01788=-62.772,-44.457,56.240,148.2344,19.3363,0.0000
C01789=-66.830,-47.084,58.128,148.1135,16.2611,0.0000
C01790=-71.379,-50.109,59.597,149.1752,10.7740,0.0000
C01791=-75.858,-52.671,60.330,157.6477,0.0531,0.0000
C01792=-80.714,-52.893,60.719,174.1606,-2.1156,0.0000
C01793=-85.269,-50.626,61.037,178.9674,-0.4701,0.0000
C01794=-88.593,-46.265,61.359,-179.8684,0.0628,0.0000
C01795=-91.197,-41.009,61.571,-179.7182,0.1356,0.0000
C01796=-93.484,-35.488,61.571,179.7049,-0.1034,0.0000
C01797=-95.359,-29.931,61.359,179.8626,-0.0486,0.0000
C01798=-96.092,-24.496,61.037,-178.9374,0.3977,0.0000
C01799=-94.474,-19.672,60.719,-174.3703,2.6245,0.0000
C01800=-90.884,-16.396,60.330,-163.8251,15.6383,0.0000
C01801=-85.905,-15.041,59.597,-165.1443,29.2171,0.0000
C01802=-80.549,-13.963,58.128,-168.8553,33.8194,0.0000
C01803=-75.822,-12.951,56.240,-171.6938,35.8302,0.0000
C01804=-72.328,-11.825,54.436,-174.0078,36.9792,0.0000
C01805=-70.362,-9.959,53.146,-176.8908,37.9934,0.0000
C01806=-69.984,-6.412,52.637,178.5225,38.8023,0.0000
C01807=-70.158,-3.072,52.615,177.6237,38.9026,0.0000
C01808=-70.224,0.000,52.630,179.9996,38.9537,0.0000
C01809=-70.158,3.071,52.615,-177.6234,38.9027,0.0000
C01810=-69.984,6.412,52.637,-178.5239,38.8022,0.0000
C01811=-70.362,9.959,53.146,176.8902,37.9933,0.0000
C01812=-72.328,11.825,54.436,174.0076,36.9792,0.0000
C01813=-75.822,12.951,56.240,171.6939,35.8303,0.0000
C01814=-80.549,13.963,58.128,168.8556,33.8196,0.0000
C01815=-85.905,15.041,59.597,165.1447,29.2176,0.0000
C01816=-90.884,16.396,60.330,163.8251,15.6386,0.0000
C01817=-94.474,19.672,60.719,174.3703,2.6245,0.0000
C01818=-96.092,24.496,61.037,178.9374,0.3977,0.0000
C01819=-95.359,29.931,61.359,-179.8626,-0.0486,0.0000
C01820=-93.484,35.488,61.571,-179.7049,-0.1034,0.0000
C01821=-91.197,41.009,61.571,179.7182,0.1356,0.0000
C01822=-88.593,46.265,61.359,179.8684,0.0628,0.0000
C01823=-85.269,50.626,61.037,-178.9674,-0.4701,0.0000
C01824=-80.714,52.893,60.719,-174.1606,-2.1156,0.0000
C01825=-75.858,52.671,60.330,-157.6479,0.0529,0.0000
C01826=-71.379,50.109,59.597,-149.1753,10.7734,0.0000
C01827=-66.830,47.084,58.128,-148.1134,16.2608,0.0000
C01828=-62.772,44.457,56.240,-148.2344,19.3362,0.0000
C01829=-59.505,42.782,54.436,-148.6339,21.4921,0.0000
C01830=-56.796,42.712,53.146,-149.3937,23.8942,0.0000
C01831=-54.020,44.952,52.637,-151.1661,27.2134,0.0000
C01832=-51.781,47.437,52.615,-151.5527,27.8318,0.0000
C01833=-49.656,49.656,52.630,-150.2454,26.3949,0.0000
C01834=-47.437,51.781,52.615,-149.0170,24.9132,0.0000
C01835=-44.952,54.020,52.637,-149.5878,25.3979,0.0000
C01836=-42.711,56.796,53.146,-152.7643,27.7428,0.0000
C01837=-42.782,59.505,54.436,-155.2436,28.9675,0.0000
C01838=-44.457,62.772,56.240,-157.5727,29.7852,0.0000
C01839=-47.084,66.830,58.128,-161.0412,30.4713,0.0000
C01840=-50.109,71.379,59.597,-167.5055,30.2239,0.0000
C01841=-52.671,75.858,60.330,-179.9426,22.3523,0.0000
C01842=-52.893,80.714,60.719,177.8734,5.8354,0.0000
C01843=-50.626,85.269,61.037,179.5298,1.0326,0.0000
C01844=-46.265,88.593,61.359,-179.9372,-0.1316,0.0000
C01845=-41.009,91.197,61.571,-179.8644,-0.2818,0.0000
C01846=-35.488,93.484,61.571,179.8966,0.2951,0.0000
C01847=-29.931,95.359,61.359,179.9514,0.1374,0.0000
C01848=-24.496,96.092,61.037,-179.6023,-1.0626,0.0000
C01849=-19.672,94.474,60.719,-177.3628,-5.6237,0.0000
C01850=-16.396,90.884,60.330,-163.7502,-15.5606,0.0000
C01851=-15.041,85.905,59.597,-149.9453,-12.9300,0.0000
C01852=-13.963,80.549,58.128,-145.6743,-9.2404,0.0000
C01853=-12.951,75.822,56.240,-143.8825,-6.7261,0.0000
C01854=-11.825,72.328,54.436,-142.8698,-4.7839,0.0000
C01855=-9.959,70.362,53.146,-141.9657,-2.4503,0.0000
C01856=-6.412,69.984,52.637,-141.1885,1.1503,0.0000
C01857=-3.071,70.158,52.615,-141.0732,1.8493,0.0000
C01858=0.000,70.224,52.630,-141.0463,-0.0003,0.0000
C01859=0.000,68.843,54.342,-141.2420,-0.0004,0.0000
C01860=2.945,68.781,54.326,-141.2681,-1.8163,0.0000
C01861=6.200,68.619,54.350,-141.3822,-1.0969,0.0000
C01862=9.699,69.044,54.888,-142.1619,2.5297,0.0000
